(* IEC 61131-3 sources: CodesysTest/export, 96 files *)

(* ---- CheckIfHomed.st ---- *)
FUNCTION CheckIfHomed : BOOL
VAR_INPUT
	Component : IComponent;
END_VAR
VAR
	homableDevice : IHomable;
END_VAR

//	Function: CheckIfHomed()
//	Description: Helper function
//				 Pass in a component - if it has a homable motor, and is not yet homed, start homing
//	Created by: Ben Hess
//	Created Date: May 16th, 2019

IF (__QUERYINTERFACE(Component, homableDevice)) THEN
	IF homableDevice.IsHomed OR NOT Component.OptionActive THEN
		CheckIfHomed := TRUE;
		RETURN;
	ELSE
		RETURN;
	END_IF
END_IF

FUNCTION CheckIfHomed : BOOL
VAR_INPUT
	Component : IComponent;
END_VAR
VAR
	homableDevice : IHomable;
END_VAR

//	Function: CheckIfHomed()
//	Description: Helper function
//				 Pass in a component - if it has a homable motor, and is not yet homed, start homing
//	Created by: Ben Hess
//	Created Date: May 16th, 2019

IF (__QUERYINTERFACE(Component, homableDevice)) THEN
	IF homableDevice.IsHomed OR NOT Component.OptionActive THEN
		CheckIfHomed := TRUE;
		RETURN;
	ELSE
		RETURN;
	END_IF
END_IF

(* ---- EnableSimulation.st ---- *)
FUNCTION EnableSimulation : BOOL
VAR_INPUT
	device : IAllObjects;
	enableSim : BOOL;
END_VAR
VAR
	simulatable : ISimulateable;
END_VAR

//	Function: EnableSimulation()
//	Description: Helper function
//				 Pass in a device. Set simulation status if possible
//	Created by: Ben Hess
//	Created Date: June 25th, 2019

IF (__QUERYINTERFACE(device, simulatable)) THEN
	simulatable.Simulate := enableSim;
END_IF

FUNCTION EnableSimulation : BOOL
VAR_INPUT
	device : IAllObjects;
	enableSim : BOOL;
END_VAR
VAR
	simulatable : ISimulateable;
END_VAR

//	Function: EnableSimulation()
//	Description: Helper function
//				 Pass in a device. Set simulation status if possible
//	Created by: Ben Hess
//	Created Date: June 25th, 2019

IF (__QUERYINTERFACE(device, simulatable)) THEN
	simulatable.Simulate := enableSim;
END_IF

(* ---- ExhaustIfPossible.st ---- *)
FUNCTION ExhaustIfPossible : BOOL  // Attempts to exhaust SV, returns true if exhaust commanded
VAR_INPUT
	device : IAllObjects;
END_VAR
VAR
	exhaustableDevice : IExhaustable;
END_VAR

//	Function: ExhaustIfPossible()
//	Description: Helper function
//				 Pass in a device that is controlled byt a SV - exhaust if possible
//	Created by: Ben Hess
//	Created Date: June 25th, 2019

IF (__QUERYINTERFACE(device, exhaustableDevice)) THEN
	exhaustableDevice.Exhaust();
	ExhaustIfPossible := TRUE;
ELSE
	ExhaustIfPossible := FALSE;
END_IF

FUNCTION ExhaustIfPossible : BOOL  // Attempts to exhaust SV, returns true if exhaust commanded
VAR_INPUT
	device : IAllObjects;
END_VAR
VAR
	exhaustableDevice : IExhaustable;
END_VAR

//	Function: ExhaustIfPossible()
//	Description: Helper function
//				 Pass in a device that is controlled byt a SV - exhaust if possible
//	Created by: Ben Hess
//	Created Date: June 25th, 2019

IF (__QUERYINTERFACE(device, exhaustableDevice)) THEN
	exhaustableDevice.Exhaust();
	ExhaustIfPossible := TRUE;
ELSE
	ExhaustIfPossible := FALSE;
END_IF

(* ---- ExtendLPIfPossible.st ---- *)
FUNCTION ExtendLPIfPossible : BOOL
VAR_INPUT
	device : IAllObjects;
END_VAR
VAR
	extendLowPressureDevice : IExtendLowPressure;
END_VAR

//	Function: ExtendLPIfPossible()
//	Description: Helper function
//				 Pass in a device that is controlled byt a SV - extend at low pressure if possible
//	Created by: Ben Hess
//	Created Date: June 27th, 2019

IF (__QUERYINTERFACE(device, extendLowPressureDevice)) THEN
	extendLowPressureDevice.ExtendLowPressure();
	ExtendLPIfPossible := TRUE;
ELSE
	ExtendLPIfPossible := FALSE;
END_IF

FUNCTION ExtendLPIfPossible : BOOL
VAR_INPUT
	device : IAllObjects;
END_VAR
VAR
	extendLowPressureDevice : IExtendLowPressure;
END_VAR

//	Function: ExtendLPIfPossible()
//	Description: Helper function
//				 Pass in a device that is controlled byt a SV - extend at low pressure if possible
//	Created by: Ben Hess
//	Created Date: June 27th, 2019

IF (__QUERYINTERFACE(device, extendLowPressureDevice)) THEN
	extendLowPressureDevice.ExtendLowPressure();
	ExtendLPIfPossible := TRUE;
ELSE
	ExtendLPIfPossible := FALSE;
END_IF

(* ---- FirstScan.st ---- *)
FUNCTION FirstScan : DWORD
VAR_IN_OUT
	EventPrm: CmpApp.EVTPARAM_CmpApp;
END_VAR
VAR
END_VAR
// Set first scan flag from StartDone system event
Globals.firstScan := TRUE;

FUNCTION FirstScan : DWORD
VAR_IN_OUT
	EventPrm: CmpApp.EVTPARAM_CmpApp;
END_VAR
VAR
END_VAR
// Set first scan flag from StartDone system event
Globals.firstScan := TRUE;

(* ---- FN_RandomDINT.st ---- *)
FUNCTION FN_RandomDINT : DINT
VAR_INPUT
	last : DINT;
	low : DINT;
	high : DINT;
END_VAR
VAR
END_VAR

FN_RandomDINT := TO_DINT(OSCAT_BASIC.RDM(OSCAT_BASIC.FRACT(TO_REAL(last) * OSCAT_BASIC.Globale_Variablen.MATH.PI)) * (TO_REAL(high) - TO_REAL(low) + 1)) + low;

FUNCTION FN_RandomDINT : DINT
VAR_INPUT
	last : DINT;
	low : DINT;
	high : DINT;
END_VAR
VAR
END_VAR

FN_RandomDINT := TO_DINT(OSCAT_BASIC.RDM(OSCAT_BASIC.FRACT(TO_REAL(last) * OSCAT_BASIC.Globale_Variablen.MATH.PI)) * (TO_REAL(high) - TO_REAL(low) + 1)) + low;

(* ---- GetBooleanProperty.st ---- *)
// This function has been automatically generated from the project information.
{attribute 'signature_flag' := '1073741824'}
{attribute 'register_in_runtime'}
FUNCTION GetBooleanProperty : BOOL
VAR_INPUT
	stKey: WSTRING;
END_VAR
GetBooleanProperty := FALSE;

(* ---- GetCompany.st ---- *)
// This function has been automatically generated from the project information.
{attribute 'signature_flag' := '1073741824'}
{attribute 'register_in_runtime'}
FUNCTION GetCompany : WSTRING
VAR_INPUT

END_VAR
GetCompany := "Sharp Packaging";

// This function has been automatically generated from the project information.
{attribute 'signature_flag' := '1073741824'}
{attribute 'register_in_runtime'}
FUNCTION GetCompany : WSTRING
VAR_INPUT

END_VAR
GetCompany := "Sharp Packaging";

(* ---- GetLibVersion.st ---- *)
// This function has been automatically generated from the project information.
FUNCTION GetLibVersion : VERSION
VAR_INPUT

END_VAR
GetLibVersion.uiMajor := 0;
GetLibVersion.uiMinor := 2;
GetLibVersion.uiServicePack := 1;
GetLibVersion.uiPatch := 122;

// This function has been automatically generated from the project information.
FUNCTION GetLibVersion : VERSION
VAR_INPUT

END_VAR
GetLibVersion.uiMajor := 0;
GetLibVersion.uiMinor := 2;
GetLibVersion.uiServicePack := 1;
GetLibVersion.uiPatch := 122;

(* ---- GetLibVersionNumber.st ---- *)
// This function has been automatically generated from the project information.
FUNCTION GetLibVersionNumber : DWORD
VAR_INPUT

END_VAR
GetLibVersionNumber := 131450;

// This function has been automatically generated from the project information.
FUNCTION GetLibVersionNumber : DWORD
VAR_INPUT

END_VAR
GetLibVersionNumber := 131450;

(* ---- GetNumberProperty.st ---- *)
// This function has been automatically generated from the project information.
{attribute 'signature_flag' := '1073741824'}
{attribute 'register_in_runtime'}
FUNCTION GetNumberProperty : DINT
VAR_INPUT
	stKey: WSTRING;
END_VAR
GetNumberProperty := 0;

(* ---- GetTextProperty.st ---- *)
// This function has been automatically generated from the project information.
{attribute 'signature_flag' := '1073741824'}
{attribute 'register_in_runtime'}
FUNCTION GetTextProperty : WSTRING
VAR_INPUT
	stKey: WSTRING;
END_VAR
IF stKey = "Company" THEN
	GetTextProperty := "Sharp Packaging";
ELSIF stKey = "Project" THEN
	GetTextProperty := "SharpBagger";
ELSIF stKey = "Title" THEN
	GetTextProperty := "Sharp Bagger";
ELSE
	GetTextProperty := "";
END_IF

// This function has been automatically generated from the project information.
{attribute 'signature_flag' := '1073741824'}
{attribute 'register_in_runtime'}
FUNCTION GetTextProperty : WSTRING
VAR_INPUT
	stKey: WSTRING;
END_VAR
IF stKey = "Company" THEN
	GetTextProperty := "Sharp Packaging";
ELSIF stKey = "Project" THEN
	GetTextProperty := "SharpBagger";
ELSIF stKey = "Title" THEN
	GetTextProperty := "Sharp Bagger";
ELSE
	GetTextProperty := "";
END_IF

(* ---- GetTitle.st ---- *)
// This function has been automatically generated from the project information.
{attribute 'signature_flag' := '1073741824'}
{attribute 'register_in_runtime'}
FUNCTION GetTitle : WSTRING
VAR_INPUT

END_VAR
GetTitle := "Sharp Bagger";

(* ---- GetVersion.st ---- *)
// This function has been automatically generated from the project information.
{attribute 'signature_flag' := '1073741824'}
{attribute 'register_in_runtime'}
FUNCTION GetVersion : VERSION
VAR_INPUT

END_VAR
GetVersion.uiMajor := 0;
GetVersion.uiMinor := 2;
GetVersion.uiServicePack := 1;
GetVersion.uiPatch := 122;

(* ---- GetVersionProperty.st ---- *)
// This function has been automatically generated from the project information.
{attribute 'signature_flag' := '1073741824'}
{attribute 'register_in_runtime'}
FUNCTION GetVersionProperty : VERSION
VAR_INPUT
	stKey: WSTRING;
END_VAR
IF stKey = "Version" THEN
	GetVersionProperty.uiMajor := 0;
	GetVersionProperty.uiMinor := 2;
	GetVersionProperty.uiServicePack := 1;
	GetVersionProperty.uiPatch := 122;
ELSE
	GetVersionProperty.uiMajor := 0;
	GetVersionProperty.uiMinor := 0;
	GetVersionProperty.uiServicePack := 0;
	GetVersionProperty.uiPatch := 0;
END_IF

// This function has been automatically generated from the project information.
{attribute 'signature_flag' := '1073741824'}
{attribute 'register_in_runtime'}
FUNCTION GetVersionProperty : VERSION
VAR_INPUT
	stKey: WSTRING;
END_VAR
IF stKey = "Version" THEN
	GetVersionProperty.uiMajor := 0;
	GetVersionProperty.uiMinor := 2;
	GetVersionProperty.uiServicePack := 1;
	GetVersionProperty.uiPatch := 122;
ELSE
	GetVersionProperty.uiMajor := 0;
	GetVersionProperty.uiMinor := 0;
	GetVersionProperty.uiServicePack := 0;
	GetVersionProperty.uiPatch := 0;
END_IF

(* ---- HomeIfNeeded.st ---- *)
FUNCTION HomeIfNeeded : BOOL
VAR_INPUT
	Component : IComponent;
END_VAR
VAR
	homableDevice : IHomable;
END_VAR

//	Function: HomeIfNeeded()
//	Description: Helper function
//				 Pass in a component - if it has a homable motor, and is not yet homed, start homing
//	Created by: Ben Hess
//	Created Date: May 16th, 2019

IF (__QUERYINTERFACE(Component, homableDevice)) AND Component.OptionActive THEN
	IF homableDevice.IsHomed THEN
		HomeIfNeeded := TRUE;
		RETURN;
	ELSE
		homableDevice.HomeNow();
	END_IF
END_IF

(* ---- IsLibReleased.st ---- *)
// This function has been automatically generated from the project information.
FUNCTION IsLibReleased : BOOL
VAR_INPUT

END_VAR
IsLibReleased := FALSE;

(* ---- MoveRequested.st ---- *)
FUNCTION MoveRequested : BOOL
VAR_INPUT
	Component : IComponent;
END_VAR
VAR
	movableDevice : IPostHomeMove;
END_VAR

//	Function: MoveIfNeeded()
//	Description: Helper function
//				 Pass in a component - if it has a homable motor, and is not yet homed, start homing
//	Created by: Ben Hess
//	Created Date: May 16th, 2019

IF (__QUERYINTERFACE(Component, movableDevice)) AND Component.OptionActive THEN
	IF NOT movableDevice.InDesiredPosition THEN
		MoveRequested := TRUE;
		RETURN;
	ELSE
		RETURN;
	END_IF
END_IF

FUNCTION MoveRequested : BOOL
VAR_INPUT
	Component : IComponent;
END_VAR
VAR
	movableDevice : IPostHomeMove;
END_VAR

//	Function: MoveIfNeeded()
//	Description: Helper function
//				 Pass in a component - if it has a homable motor, and is not yet homed, start homing
//	Created by: Ben Hess
//	Created Date: May 16th, 2019

IF (__QUERYINTERFACE(Component, movableDevice)) AND Component.OptionActive THEN
	IF NOT movableDevice.InDesiredPosition THEN
		MoveRequested := TRUE;
		RETURN;
	ELSE
		RETURN;
	END_IF
END_IF

(* ---- MoveTimeoutCalc.st ---- *)
FUNCTION MoveTimeoutCalc : TIME
VAR_INPUT
	distance : REAL;
	velo : REAL;
	buffer : REAL;		// Buffer time to add for timeout
END_VAR
VAR
END_VAR

MoveTimeoutCalc := TO_TIME(((ABS(distance) / velo) * 1000) + buffer);

(* ---- PostHomeMoveIfNeeded.st ---- *)
FUNCTION PostHomeMoveIfNeeded : BOOL
VAR_INPUT
	Component : IComponent;
END_VAR
VAR
	movableDevice : IPostHomeMove;
END_VAR

//	Function: MoveIfNeeded()
//	Description: Helper function
//				 Pass in a component - if it has a homable motor, and is homed, and is configured for a post homing move, perform it
//	Created by: Ben Hess
//	Created Date: May 16th, 2019

IF (__QUERYINTERFACE(Component, movableDevice)) AND Component.OptionActive THEN
	IF movableDevice.InDesiredPosition THEN
		PostHomeMoveIfNeeded := TRUE;
		RETURN;
	ELSE
		movableDevice.MoveNow();
	END_IF
END_IF

(* ---- EM01_Bagger_Control_Modules.st ---- *)
FUNCTION_BLOCK EM01_Bagger_Control_Modules
VAR_INPUT
END_VAR
VAR_OUTPUT

	//simBagDelivery : FB_SimBasicBagDelivery(name := 'Sim Bag Delivery'):= (enable := TRUE, installed := TRUE);
	//simPrinter : FB_SimBasicPrinter(name := 'Sim Printer'):= (enable := TRUE, installed := TRUE);
	//simVacuumCups : FB_SimBasicVacuum(name := 'Sim Vac Cups') := (_optionEnabled := TRUE, _optionInstalled := TRUE);
	vacuumCups : FB_PneumaticVacuumCups(name := 'Pneumatic Vacuum Cups') := (_optionEnabled := TRUE, _optionInstalled := TRUE);
	simLoadPlate : FB_SimBasicLoadPlate(name := 'Sim Load Plate') := (_optionEnabled := TRUE, _optionInstalled := TRUE);
	simExitConveyor : FB_SimBasicExitConveyor(name := 'Sim Exit Conveyor') := (_optionEnabled := TRUE, _optionInstalled := TRUE);

	standardSealBar : FB_PneumaticSealer(name := 'Pneumatic Seal Bar') := (_optionEnabled := TRUE, _optionInstalled := TRUE);
	standardBagOpenFingersWithSensors : FB_PneuBagOpenFingersWithSensorsOLD(name := 'Standard Bag Open Fingers') := (_optionEnabled := TRUE, _optionInstalled := TRUE);
	pneumaticPressureBar : FB_PneuPBarWithAdjPass(name := 'Pneumatic Pressure Bar') := (_optionEnabled := TRUE, _optionInstalled := TRUE);
	motorizedSealFlatteners : FB_MotorizedSealFlatteners(name := 'Motorized Seal Flatteners') := (_optionEnabled := TRUE, _optionInstalled := TRUE);

	passthroughMotor : FB_SimMotor;
	msfHorizontalMotor : FB_SimMotor;
	bagOpenFingersActuator : FB_PneumaticVerticalActuator(name := 'Bag Open Fingers Actuator');
	sealFlattenerVertAxisActuator : FB_PneumaticVerticalActuator(name := 'Seal Flat Pneu Vert Axis Actuator');

	bagDelivery : FB_Pro18BagDelivery(name := 'Bag Delivery') := (_optionEnabled := TRUE, _optionInstalled := TRUE);
	bagDeliveryFrontMotor : FB_SimMotor;

	labelPrinter : FB_Pro18ZebraPrinter(name := 'Zebra Label Printer') := (_optionEnabled := TRUE, _optionInstalled := TRUE);
	printHeadActuator : FB_PneumaticVerticalActuator(name := 'Print Head Actuator');
END_VAR

VAR
END_VAR

// simBagDelivery(
// 	enable:= ,
// 	installed:= ,
// 	active=> ,
// 	feedSpeed:= HMI.data.bagForwardSpeed,
// 	reverseSpeed:= HMI.data.bagReverseSpeed,
// 	printSpeed:= HMI.data.printSpeed,
// 	printLength:= HMI.data.printLength,
// 	bagLength:= HMI.data.bagLength,
// 	reverseLength:= 2.0,
// 	printOffset:= HMI.data.printOffset);

//sealFlattenerPneuVerticalAxis(cylinder := sealFlattenerVertAxisActuator);

simExitConveyor(_optionActive=> );

simLoadPlate(_optionActive=> , loadPlateDwell:= HMI.data.loadPlateDwell);

passthroughMotor(simFault := UN00_Globals.simFaults.passthroughMotorFault);

pneumaticPressureBar(
	_optionActive=> ,
	simulateIO:= HMI.data.simulateAllIO,
	passthroughMotor:= passthroughMotor,
	cylinder := Devices.pressureBarSolenoidValve,
	ptVelo:= ,
	ptAccel:= ,
	ptDecel:= ,
	homeTimeoutSetting:= ,
	passthroughSetting := HMI.data.passthroughSetting,
	failedToClose=> ,
	failedToOpen=> ,
	failedToHome=> ,
	pressureBarObstructed=> ,
	motorFault=> ,
	failedToMovePassthrough=> ,
	actualPassthrough=> HMI.data.passthroughActual,
	PressureBarClosedSensor:= IO.iPressureBarRetracted,
	PressureBarOpenSensor:= IO.iPressureBarExtended,
	ObstructionSensor := IO.iPressureBarNotObstructed);

printHeadActuator(cylinder := Devices.printHeadSolenoidValve);
labelPrinter(
	_optionActive=> ,
	simulateIO:= HMI.data.simulateAllIO,
	printSpeed:= HMI.data.printSpeed,
	printLength:= HMI.data.printLength,
	printHead:= printHeadActuator,
	dataReadyInput:= IO.iPrinterDataReady,
	serviceRequiredInput:= IO.iPrinterServiceRequired,
	ribbonLowInput:= IO.iPrinterRibbonOut,
	endOfPrintInput:= IO.iPrinterEndOfPrint,
	printHeadDebounceSetpoint:= ,
	serviceRequired=> ,
	ribbonLow=> ,
	startPrintOutput:= IO.oPrinterStartPrint,
	ribbonUnwindRunOutput:= IO.oRunRibbonUnwindMotor);

standardSealBar(
	_optionActive=> ,
	simulateIO:= HMI.data.simulateAllIO,
	sealDwell:= HMI.data.sealBarDwell,
	cylinder:= Devices.sealBarSolenoidValve);

vacuumCups(_optionActive=>, vacGenerator := Devices.vacuumSolenoidValve);
bagOpenFingersActuator(cylinder:= Devices.bagOpenFingersSolenoidValve);
standardBagOpenFingersWithSensors(
	simulateIO:= HMI.data.simulateAllIO,
	simMissedBag:= UN00_Globals.simFaults.failedToGrabBagLeftFinger,
	_optionActive=> ,
	delayToGrabSetting:= HMI.data.grabBagDelay,
	delayToCheckBagPresentSetting:= HMI.data.checkForBagOpenDelay,
	delayToClearSetting:= HMI.data.bagClearedFromFingersDelay,
	fingerActuators := bagOpenFingersActuator,
	BagPresentSensorLeft:= IO.iBagOpenFingersLeftBagPresent,
	BagPresentSensorRight:= IO.iBagOpenFingersRightBagPresent);

sealFlattenerVertAxisActuator(solenoid0=> , solenoid1=> , cylinder:= Devices.sealFlattenersVertAxisSolenoidValve);
msfHorizontalMotor();
motorizedSealFlatteners(
	_optionActive=> ,
	clearanceDwellSetting:= HMI.data.bagDropClearanceDwell,
	bagWidth:= HMI.data.bagWidth,
	horizVelo:= ,
	horizAccel:= ,
	horizDecel:= ,
	bagHoldingCurrent:= ,
	sealCurrentAddition:= ,
	homeTimeoutSetting:= ,
	maximumPosition:= ,
	miniumumPosition:= ,
	clearanceOffset:= ,
	msfHorizActualPosition=> ,
	horizontalFailedToMove=> ,
	horizontalFailedToHome=> ,
	motorFault=> ,
	verticalAxis:= sealFlattenerVertAxisActuator,
	horizontalAxis:= msfHorizontalMotor);

	bagDeliveryFrontMotor();
	bagDelivery(
	simulateIO := HMI.data.simulateAllIO,
	_optionActive=> ,
	printer:= labelPrinter,
	bagLength:= HMI.data.bagLength,
	feedSpeed:= TO_REAL(HMI.data.bagForwardSpeed),
	reverseSpeed:= TO_REAL(HMI.data.bagReverseSpeed),
	printSpeed:= ,
	printOffset:= ,
	printLength:= ,
	maxReverseSetpoint:= ,
	sealOffset:= ,
	distanceFromSealBarToBagEdge:= ,
	distanceFromNipToBagEdge:= ,
	bagPhotoeyeInput:= IO.iBagPhotoeyeClear,
	trapezoidalPercent:= ,
	bagDeliveryFailedToMove=> ,
	bagFailedToSeparate=> ,
	bagDeliveryMotor:= bagDeliveryFrontMotor);

FUNCTION_BLOCK EM01_Bagger_Control_Modules
VAR_INPUT
END_VAR
VAR_OUTPUT

	//simBagDelivery : FB_SimBasicBagDelivery(name := 'Sim Bag Delivery'):= (enable := TRUE, installed := TRUE);
	//simPrinter : FB_SimBasicPrinter(name := 'Sim Printer'):= (enable := TRUE, installed := TRUE);
	//simVacuumCups : FB_SimBasicVacuum(name := 'Sim Vac Cups') := (_optionEnabled := TRUE, _optionInstalled := TRUE);
	vacuumCups : FB_PneumaticVacuumCups(name := 'Pneumatic Vacuum Cups') := (_optionEnabled := TRUE, _optionInstalled := TRUE);
	simLoadPlate : FB_SimBasicLoadPlate(name := 'Sim Load Plate') := (_optionEnabled := TRUE, _optionInstalled := TRUE);
	simExitConveyor : FB_SimBasicExitConveyor(name := 'Sim Exit Conveyor') := (_optionEnabled := TRUE, _optionInstalled := TRUE);

	standardSealBar : FB_PneumaticSealer(name := 'Pneumatic Seal Bar') := (_optionEnabled := TRUE, _optionInstalled := TRUE);
	standardBagOpenFingersWithSensors : FB_PneuBagOpenFingersWithSensorsOLD(name := 'Standard Bag Open Fingers') := (_optionEnabled := TRUE, _optionInstalled := TRUE);
	pneumaticPressureBar : FB_PneuPBarWithAdjPass(name := 'Pneumatic Pressure Bar') := (_optionEnabled := TRUE, _optionInstalled := TRUE);
	motorizedSealFlatteners : FB_MotorizedSealFlatteners(name := 'Motorized Seal Flatteners') := (_optionEnabled := TRUE, _optionInstalled := TRUE);

	passthroughMotor : FB_SimMotor;
	msfHorizontalMotor : FB_SimMotor;
	bagOpenFingersActuator : FB_PneumaticVerticalActuator(name := 'Bag Open Fingers Actuator');
	sealFlattenerVertAxisActuator : FB_PneumaticVerticalActuator(name := 'Seal Flat Pneu Vert Axis Actuator');

	bagDelivery : FB_Pro18BagDelivery(name := 'Bag Delivery') := (_optionEnabled := TRUE, _optionInstalled := TRUE);
	bagDeliveryFrontMotor : FB_SimMotor;

	labelPrinter : FB_Pro18ZebraPrinter(name := 'Zebra Label Printer') := (_optionEnabled := TRUE, _optionInstalled := TRUE);
	printHeadActuator : FB_PneumaticVerticalActuator(name := 'Print Head Actuator');
END_VAR

VAR
END_VAR

// simBagDelivery(
// 	enable:= ,
// 	installed:= ,
// 	active=> ,
// 	feedSpeed:= HMI.data.bagForwardSpeed,
// 	reverseSpeed:= HMI.data.bagReverseSpeed,
// 	printSpeed:= HMI.data.printSpeed,
// 	printLength:= HMI.data.printLength,
// 	bagLength:= HMI.data.bagLength,
// 	reverseLength:= 2.0,
// 	printOffset:= HMI.data.printOffset);

//sealFlattenerPneuVerticalAxis(cylinder := sealFlattenerVertAxisActuator);

simExitConveyor(_optionActive=> );

simLoadPlate(_optionActive=> , loadPlateDwell:= HMI.data.loadPlateDwell);

passthroughMotor(simFault := UN00_Globals.simFaults.passthroughMotorFault);

pneumaticPressureBar(
	_optionActive=> ,
	simulateIO:= HMI.data.simulateAllIO,
	passthroughMotor:= passthroughMotor,
	cylinder := Devices.pressureBarSolenoidValve,
	ptVelo:= ,
	ptAccel:= ,
	ptDecel:= ,
	homeTimeoutSetting:= ,
	passthroughSetting := HMI.data.passthroughSetting,
	failedToClose=> ,
	failedToOpen=> ,
	failedToHome=> ,
	pressureBarObstructed=> ,
	motorFault=> ,
	failedToMovePassthrough=> ,
	actualPassthrough=> HMI.data.passthroughActual,
	PressureBarClosedSensor:= IO.iPressureBarRetracted,
	PressureBarOpenSensor:= IO.iPressureBarExtended,
	ObstructionSensor := IO.iPressureBarNotObstructed);

printHeadActuator(cylinder := Devices.printHeadSolenoidValve);
labelPrinter(
	_optionActive=> ,
	simulateIO:= HMI.data.simulateAllIO,
	printSpeed:= HMI.data.printSpeed,
	printLength:= HMI.data.printLength,
	printHead:= printHeadActuator,
	dataReadyInput:= IO.iPrinterDataReady,
	serviceRequiredInput:= IO.iPrinterServiceRequired,
	ribbonLowInput:= IO.iPrinterRibbonOut,
	endOfPrintInput:= IO.iPrinterEndOfPrint,
	printHeadDebounceSetpoint:= ,
	serviceRequired=> ,
	ribbonLow=> ,
	startPrintOutput:= IO.oPrinterStartPrint,
	ribbonUnwindRunOutput:= IO.oRunRibbonUnwindMotor);

standardSealBar(
	_optionActive=> ,
	simulateIO:= HMI.data.simulateAllIO,
	sealDwell:= HMI.data.sealBarDwell,
	cylinder:= Devices.sealBarSolenoidValve);

vacuumCups(_optionActive=>, vacGenerator := Devices.vacuumSolenoidValve);
bagOpenFingersActuator(cylinder:= Devices.bagOpenFingersSolenoidValve);
standardBagOpenFingersWithSensors(
	simulateIO:= HMI.data.simulateAllIO,
	simMissedBag:= UN00_Globals.simFaults.failedToGrabBagLeftFinger,
	_optionActive=> ,
	delayToGrabSetting:= HMI.data.grabBagDelay,
	delayToCheckBagPresentSetting:= HMI.data.checkForBagOpenDelay,
	delayToClearSetting:= HMI.data.bagClearedFromFingersDelay,
	fingerActuators := bagOpenFingersActuator,
	BagPresentSensorLeft:= IO.iBagOpenFingersLeftBagPresent,
	BagPresentSensorRight:= IO.iBagOpenFingersRightBagPresent);

sealFlattenerVertAxisActuator(solenoid0=> , solenoid1=> , cylinder:= Devices.sealFlattenersVertAxisSolenoidValve);
msfHorizontalMotor();
motorizedSealFlatteners(
	_optionActive=> ,
	clearanceDwellSetting:= HMI.data.bagDropClearanceDwell,
	bagWidth:= HMI.data.bagWidth,
	horizVelo:= ,
	horizAccel:= ,
	horizDecel:= ,
	bagHoldingCurrent:= ,
	sealCurrentAddition:= ,
	homeTimeoutSetting:= ,
	maximumPosition:= ,
	miniumumPosition:= ,
	clearanceOffset:= ,
	msfHorizActualPosition=> ,
	horizontalFailedToMove=> ,
	horizontalFailedToHome=> ,
	motorFault=> ,
	verticalAxis:= sealFlattenerVertAxisActuator,
	horizontalAxis:= msfHorizontalMotor);

	bagDeliveryFrontMotor();
	bagDelivery(
	simulateIO := HMI.data.simulateAllIO,
	_optionActive=> ,
	printer:= labelPrinter,
	bagLength:= HMI.data.bagLength,
	feedSpeed:= TO_REAL(HMI.data.bagForwardSpeed),
	reverseSpeed:= TO_REAL(HMI.data.bagReverseSpeed),
	printSpeed:= ,
	printOffset:= ,
	printLength:= ,
	maxReverseSetpoint:= ,
	sealOffset:= ,
	distanceFromSealBarToBagEdge:= ,
	distanceFromNipToBagEdge:= ,
	bagPhotoeyeInput:= IO.iBagPhotoeyeClear,
	trapezoidalPercent:= ,
	bagDeliveryFailedToMove=> ,
	bagFailedToSeparate=> ,
	bagDeliveryMotor:= bagDeliveryFrontMotor);

(* ---- EM01_BaggerHead.st ---- *)
FUNCTION_BLOCK EM01_BaggerHead EXTENDS FB_PackMLStates IMPLEMENTS IEM01_BaggerHead
VAR_INPUT
	(*Comnponents*)
	bagOpenFingers : IBagOpenFingers;
	sealFlatteners : ISealFlatteners;
	sealer : ISealer;
	pressureBar : IPressureBar;
	printer : IPrinter;
	bagDelivery : IBagDelivery;
	vacuumBagOpen : IVacuumBagOpen;

	(*Options and settings*)
	bagOpenAssistEnabled : BOOL;		// Bag Open Assist Option Enabled from HMI
	bagOpenSensorEnabled : BOOL;		// Bag Open Sensors Enabled from HMI
	separateBeforeSealEnabled : BOOL;	// Separate before Seal Option Enabled from HMI
	bagOpenRetrySetting : UINT;
	newJobLoaded : BOOL;
	vacuumDwell : TIME;
END_VAR
VAR_OUTPUT
	baggerCycleActive : BOOL;
	bagOpenRetryCount : UINT;
	failedToOpenBag : FB_Fault(name := CONCAT(_prefix,'Failed to Open Bag'));
END_VAR
VAR
	_startCycle : BOOL;
	_readyToAcceptProduct : BOOL;
END_VAR

PROPERTY ReadyForProduct : BOOL

METHOD StartCycle

_startCycle := TRUE;

PROPERTY StartCycleRequest : BOOL

PROPERTY CurrentBagOpenRetryCount : UINT

FUNCTION_BLOCK EM01_BaggerHead EXTENDS FB_PackMLStates IMPLEMENTS IEM01_BaggerHead
VAR_INPUT
	(*Comnponents*)
	bagOpenFingers : IBagOpenFingers;
	sealFlatteners : ISealFlatteners;
	sealer : ISealer;
	pressureBar : IPressureBar;
	printer : IPrinter;
	bagDelivery : IBagDelivery;
	vacuumBagOpen : IVacuumBagOpen;

	(*Options and settings*)
	bagOpenAssistEnabled : BOOL;		// Bag Open Assist Option Enabled from HMI
	bagOpenSensorEnabled : BOOL;		// Bag Open Sensors Enabled from HMI
	separateBeforeSealEnabled : BOOL;	// Separate before Seal Option Enabled from HMI
	bagOpenRetrySetting : UINT;
	newJobLoaded : BOOL;
	vacuumDwell : TIME;
END_VAR
VAR_OUTPUT
	baggerCycleActive : BOOL;
	bagOpenRetryCount : UINT;
	failedToOpenBag : FB_Fault(name := CONCAT(_prefix,'Failed to Open Bag'));
END_VAR
VAR
	_startCycle : BOOL;
	_readyToAcceptProduct : BOOL;
END_VAR

PROPERTY ReadyForProduct : BOOL

METHOD StartCycle

_startCycle := TRUE;

PROPERTY StartCycleRequest : BOOL

PROPERTY CurrentBagOpenRetryCount : UINT

(* ---- EM01_BaggerHead_Automode.st ---- *)
FUNCTION_BLOCK EM01_BaggerHead_Automode EXTENDS FB_PackMLStates
VAR_INPUT
	infeed : IEM00_Product_Infeed;
	discharge : IEM02_Discharge;
END_VAR
VAR_OUTPUT
	state : HEAD_STATES;
    sealAndSeparateSubState : SEAL_SEPARATE_STATES;
    releaseAndFeedSubState : RELEASE_FEED_STATES;
    bagOpenSubState : BAG_OPEN_ASSIST_STATES;
	currentBaggerState : STRING;
END_VAR
VAR
	cycleTimer : TON() := (PT := T#1000S);
	cycleTime : REAL;
	resetTriggered : BOOL;
	resettingState : INT;
	vacuumDwellTimer : TON;
END_VAR
VAR_IN_OUT
	bagger : EM01_BaggerHead;
END_VAR

//	Function Block: EM01_Bagger_Automode
//	Description: This is an implementation of a bagger in Auto Mode (normal operation) using the PackML standard.
//				 Each method is a PackML state.
//	Created by: Ben Hess
//	Created Date: Tuesday, March 26, 2019

METHOD Stopping

_stoppingDone := TRUE;

METHOD Stopped

_clearingDone := FALSE;
_stoppingDone := FALSE;
resetTriggered := FALSE;

METHOD Resetting

state := HEAD_STATES.Idle;
sealAndSeparateSubState := SEAL_SEPARATE_STATES.Idle;
releaseAndFeedSubState := RELEASE_FEED_STATES.Idle;
bagOpenSubState := BAG_OPEN_ASSIST_STATES.Idle;

CASE resettingState OF
	0:	// Clear PackML state bits and Home everything that needs homing
		_clearingDone := FALSE;
		_completingDone := FALSE;
		_holdingDone := FALSE;
		_resettingDone := FALSE;
		_startingDone := FALSE;
		_unholdingDone := FALSE;
		_stoppingDone := FALSE;

		vacuumDwellTimer.IN := FALSE;

		bagger.bagDelivery.Reset();
		HomeIfNeeded(bagger.pressureBar);
		HomeIfNeeded(bagger.sealFlatteners);
		resettingState := 1;

	1:	// Move everything into place to start machine
		IF CheckIfHomed(bagger.pressureBar) THEN
			PostHomeMoveIfNeeded(bagger.pressureBar);
			resettingState := 2;
		END_IF

	2:	// Once everything is moved into position and ready move on
		IF bagger.pressureBar.Ready OR NOT bagger.pressureBar.OptionActive THEN
			_resettingDone := TRUE;
		END_IF

END_CASE

METHOD Idle

_resettingDone := FALSE;
resettingState := 0;
resetTriggered := FALSE;

METHOD Starting

IF NOT _startingDone THEN
	bagger.pressureBar.Open();
	bagger.bagOpenFingers.ReleaseBag();
	bagger.sealFlatteners.ToBagFeed();
	_startingDone := TRUE;
END_IF

METHOD Executing

//	Method: EM01_Bagger_Automode.Executing()
//	Description: Executing is the state in which the machine is producing bags.  In this state, the bagger is homed and ready to initiate a cycle any time.
//				 In normal operation, the machine should be in this state most of the time
//				 The logic below is generic and coded to interfaces for each component
//	Created by: Ben Hess
//	Created Date: Tuesday, March 26, 2019

IF NOT __ISVALIDREF(bagger) THEN
	RETURN;
END_IF

// Clear starting done status because if we're here starting state is complete.
_startingDone := FALSE;

// Run Cycle timer for machine cycle
cycleTimer();
vacuumDwellTimer(PT := bagger.vacuumDwell);
// State machine for overall head states
CASE state OF
    HEAD_STATES.Idle :                              // Start cycle
                                                    IF bagger.StartCycleRequest THEN
														bagger.StartCycleRequest := FALSE;
														cycleTimer.IN := TRUE;
														_logger.AddLogItem('Cycle Started');
														SetHeadState(HEAD_STATES.SealAndSeparateBag);
													END_IF

													IF MoveRequested (bagger.pressureBar) THEN
														SetHeadState(HEAD_STATES.MovePassthrough);
													END_IF

	HEAD_STATES.MovePassthrough : 					//
													PostHomeMoveIfNeeded(bagger.pressureBar);
													SetHeadState(HEAD_STATES.MovingPassthrough);

    HEAD_STATES.MovingPassthrough :                 //
													IF NOT MoveRequested (bagger.pressureBar) THEN
														SetHeadState(HEAD_STATES.MovedPassthrough);
													END_IF

	HEAD_STATES.MovedPassthrough : 					//
													SetHeadState(HEAD_STATES.Idle);

    HEAD_STATES.SealAndSeparateBag :                // Begin Seal and Separate State machine
                                                    SetSealSeparateState(SEAL_SEPARATE_STATES.MoveJawIn);
													SetHeadState(HEAD_STATES.SealingAndSeparatingBag);

    HEAD_STATES.SealingAndSeparatingBag :          //
													IF sealAndSeparateSubState = SEAL_SEPARATE_STATES.Done THEN
														SetHeadState(HEAD_STATES.SealedAndSeparatedBag);
														SetSealSeparateState(SEAL_SEPARATE_STATES.Idle);
                                                    END_IF

    HEAD_STATES.SealedAndSeparatedBag :             //
													SetHeadState(HEAD_STATES.ReleaseAndFeedBag);

    HEAD_STATES.ReleaseAndFeedBag :                 // Open the jaw and release the bag
													SetReleaseFeedState(RELEASE_FEED_STATES.MoveJawOutAndFeedBag);
                                                    SetHeadState(HEAD_STATES.ReleasingAndFeedingBag);

    HEAD_STATES.ReleasingAndFeedingBag :            //
                                                    IF releaseAndFeedSubState = RELEASE_FEED_STATES.Done THEN
                                                        SetHeadState(HEAD_STATES.ReleasedAndFedBag);
                                                        SetReleaseFeedState(RELEASE_FEED_STATES.Idle);
                                                    END_IF

    HEAD_STATES.ReleasedAndFedBag :                 // Start opening bag if bag open assist is enabled, otherwise end cycle now
													IF bagger.bagOpenAssistEnabled THEN
														SetHeadState(HEAD_STATES.OpenBag);
													ELSE
														SetHeadState(HEAD_STATES.OpenedBag);
													END_IF

    HEAD_STATES.OpenBag :                            // Close jaw to grab the bag
                                                    SetBagOpenState(BAG_OPEN_ASSIST_STATES.MoveJawIn);
                                                    SetHeadState(HEAD_STATES.OpeningBag);

    HEAD_STATES.OpeningBag :                        // Open jaw and grab onto the bag.  Feed a new bag out if missed
                                                    IF bagOpenSubState = BAG_OPEN_ASSIST_STATES.Done THEN
                                                        SetHeadState(HEAD_STATES.OpenedBag);
                                                        SetBagOpenState(BAG_OPEN_ASSIST_STATES.Idle);
													ELSIF bagOpenSubState = BAG_OPEN_ASSIST_STATES.FeedNewBag THEN
														SetHeadState(HEAD_STATES.SealAndSeparateBag);
														SetBagOpenState(BAG_OPEN_ASSIST_STATES.Idle);
                                                    END_IF

    HEAD_STATES.OpenedBag :                         // End cycle
                                                    SetHeadState(HEAD_STATES.Idle);
													cycleTime := (TIME_TO_REAL(cycleTimer.ET) / 1000);
													cycleTimer.IN := FALSE;
													_logger.AddLogItem(CONCAT('Cycle Complete in ',TO_STRING(cycleTime)));

    //HEAD_STATES.Fault :

END_CASE

CASE sealAndSeparateSubState OF
    //SEAL_SEPARATE_STATES.Idle :

    SEAL_SEPARATE_STATES.MoveJawIn :                // Perform actions as enabled - close jaw and move flatteners out. If jaw is disabled then go right to reverse bag
                                                    IF bagger.sealFlatteners.OptionActive THEN
														bagger.sealFlatteners.ToSeal();
													END_IF
                                                    bagger.pressureBar.Close();
													SetSealSeparateState(SEAL_SEPARATE_STATES.MovingJawIn);

    SEAL_SEPARATE_STATES.MovingJawIn :              // If Jaw is in and flatteners out then move on
                                                   	IF (NOT bagger.sealFlatteners.OptionActive OR bagger.sealFlatteners.InPosition)
														AND bagger.pressureBar.IsFullyClosed THEN
															SetSealSeparateState(SEAL_SEPARATE_STATES.MovedJawIn);
                                                    END_IF

    SEAL_SEPARATE_STATES.MovedJawIn :               // Seal bag now if separate before seal option selected
													IF NOT bagger.separateBeforeSealEnabled THEN
														bagger.sealer.BeginSealing();
													END_IF
													SetSealSeparateState(SEAL_SEPARATE_STATES.ReverseBag);

    SEAL_SEPARATE_STATES.ReverseBag :               // Start reversing bag to seal
													bagger.bagDelivery.ReverseToSeparate();
													SetSealSeparateState(SEAL_SEPARATE_STATES.ReversingBag);

    SEAL_SEPARATE_STATES.ReversingBag :             //
                                                    IF bagger.bagDelivery.BagSeparated
														AND (bagger.sealer.SealComplete OR bagger.separateBeforeSealEnabled)
                                                        THEN
															SetSealSeparateState(SEAL_SEPARATE_STATES.Reversedbag);
                                                    END_IF

    SEAL_SEPARATE_STATES.Reversedbag :              //
                                                    IF bagger.separateBeforeSealEnabled THEN
														SetSealSeparateState(SEAL_SEPARATE_STATES.SealBag);
													ELSE
														SetSealSeparateState(SEAL_SEPARATE_STATES.Done);
													END_IF

	SEAL_SEPARATE_STATES.SealBag:
													bagger.sealer.BeginSealing();
													SetSealSeparateState(SEAL_SEPARATE_STATES.SealingBag);

	SEAL_SEPARATE_STATES.SealingBag:				//
													IF bagger.sealer.SealComplete THEN
														SetSealSeparateState(SEAL_SEPARATE_STATES.Done);
													END_IF

    //SEAL_SEPARATE_STATES.Done :                   //

    //SEAL_SEPARATE_STATES.Fault :					//
END_CASE

CASE releaseAndFeedSubState OF
    //RELEASE_FEED_STATES.Idle :                    //

    RELEASE_FEED_STATES.MoveJawOutAndFeedBag :
													bagger.bagOpenFingers.ReleaseBag();
													bagger.sealFlatteners.ToBagFeed();
													bagger.pressureBar.Open();

													discharge.TakeAwayBag(THIS^);
													releaseAndFeedSubState := RELEASE_FEED_STATES.WaitForOKFromDischarge;
													// If printer is enabled then perform printer operation of bag delivery, otherwise just feed new bag out.
													IF NOT bagger.printer.OptionActive THEN
														bagger.bagDelivery.FeedBagOut();
														SetReleaseFeedState(RELEASE_FEED_STATES.MovingJawOutAndFeedingBag);
													ELSE
														SetReleaseFeedState(RELEASE_FEED_STATES.WaitForPrinter);
													END_IF

    RELEASE_FEED_STATES.WaitForOKFromDischarge :   	// Wait for EM02 - Discharge to give OK to feed bag signal
													IF discharge.OKToFeedBag THEN
														IF NOT bagger.printer.OptionActive THEN
															bagger.bagDelivery.FeedBagOut();
															SetReleaseFeedState(RELEASE_FEED_STATES.MovingJawOutAndFeedingBag);
														ELSE
															SetReleaseFeedState(RELEASE_FEED_STATES.WaitForPrinter);
														END_IF
													END_IF

    RELEASE_FEED_STATES.WaitForPrinter :            // Data Ready means the printer has a label and we're all set to print
                                                    IF bagger.printer.HasLabel THEN
														SetReleaseFeedState(RELEASE_FEED_STATES.FeedToOffset);
                                                    END_IF

    RELEASE_FEED_STATES.FeedToOffset :              // Start feeding to the print offset
                                                    bagger.bagDelivery.FeedToPrintOffset();
													SetReleaseFeedState(RELEASE_FEED_STATES.FeedingToOffset);

    RELEASE_FEED_STATES.FeedingToOffset :            // Once offset done start printing
                                                    IF bagger.bagDelivery.ReadyForPrint THEN
														SetReleaseFeedState(RELEASE_FEED_STATES.StartPrinting);
                                                    END_IF

    RELEASE_FEED_STATES.StartPrinting :             // Printer starts print cycle and bag delivery starts moving at print speed
													bagger.printer.BeginPrinting();
													bagger.bagDelivery.FeedAtPrintSpeed();
													SetReleaseFeedState(RELEASE_FEED_STATES.Printing);

    //RELEASE_FEED_STATES.SendPrintSignal:            //

    RELEASE_FEED_STATES.Printing :                  // Wait for print to finish
                                                    IF bagger.printer.PrintDone THEN
														SetReleaseFeedState(RELEASE_FEED_STATES.StopPrinting);
                                                    END_IF

    RELEASE_FEED_STATES.StopPrinting :              // Tell bag delivery it's okay to feed out the rest of the bag and the printer that it can prep itself for the next print
                                                    bagger.bagDelivery.FeedBagOut();
													SetReleaseFeedState(RELEASE_FEED_STATES.MovingJawOutAndFeedingBag);

    RELEASE_FEED_STATES.MovingJawOutAndFeedingBag : //
													IF (bagger.sealFlatteners.InPosition OR NOT bagger.sealFlatteners.OptionActive)
                                                        AND bagger.pressureBar.IsFullyOpen
														AND bagger.bagDelivery.BagFeedDone
                                                        THEN
															SetReleaseFeedState(RELEASE_FEED_STATES.MovedJawOutAndFedBag);
                                                    END_IF

    RELEASE_FEED_STATES.MovedJawOutAndFedBag :
													SetReleaseFeedState(RELEASE_FEED_STATES.Done);
    //RELEASE_FEED_STATES.Done :
    //RELEASE_FEED_STATES.Fault :
END_CASE

CASE bagOpenSubState OF
    BAG_OPEN_ASSIST_STATES.Idle :                    //

    BAG_OPEN_ASSIST_STATES.MoveJawIn :                // Close jaw against bag. In the future we may also start vacuum here
                                                    bagger.pressureBar.Close();
													SetBagOpenState(BAG_OPEN_ASSIST_STATES.MovingJawIn);

    BAG_OPEN_ASSIST_STATES.MovingJawIn :            // Move on once jaw is closed
                                                    IF bagger.pressureBar.IsFullyClosed THEN
														IF bagger.vacuumBagOpen.OptionActive THEN
															bagger.vacuumBagOpen.StartVacuum();
														END_IF
														SetBagOpenState(BAG_OPEN_ASSIST_STATES.MovedJawIn);
                                                    END_IF

    BAG_OPEN_ASSIST_STATES.MovedJawIn :             // Hold onto the bag with vacuum to build suction
													vacuumDwellTimer.IN := TRUE;
													IF (vacuumDwellTimer.Q OR NOT bagger.vacuumBagOpen.OptionActive) THEN
														vacuumDwellTimer.IN := FALSE;
														SetBagOpenState(BAG_OPEN_ASSIST_STATES.MoveJawOut);
													END_IF

    BAG_OPEN_ASSIST_STATES.MoveJawOut :             // Open the jaw and move seal flatteners in and to bag holding
                                                    bagger.pressureBar.Open();
													SetBagOpenState(BAG_OPEN_ASSIST_STATES.MovingJawOutAndGrab);

    BAG_OPEN_ASSIST_STATES.MovingJawOutAndGrab :    	//
														IF bagger.bagOpenFingers.OptionActive THEN
															bagger.bagOpenFingers.GrabBag();
															IF bagger.bagOpenSensorEnabled THEN
																SetBagOpenState(BAG_OPEN_ASSIST_STATES.CheckForSuccessfulBagGrab);
															ELSE
																SetBagOpenState(BAG_OPEN_ASSIST_STATES.BagOpened);
															END_IF
														ELSE
															SetBagOpenState(BAG_OPEN_ASSIST_STATES.BagOpened);
														END_IF

	BAG_OPEN_ASSIST_STATES.CheckForSuccessfulBagGrab : 	//
														IF bagger.CurrentBagOpenRetryCount < bagger.bagOpenRetrySetting THEN
															IF bagger.bagOpenFingers.BagGrabbed THEN
																SetBagOpenState(BAG_OPEN_ASSIST_STATES.BagOpened);
															ELSIF bagger.bagOpenFingers.BagMissed THEN
																SetBagOpenState(BAG_OPEN_ASSIST_STATES.BagFailedToOpen);
															END_IF
														ELSE
															SetBagOpenState(BAG_OPEN_ASSIST_STATES.MovingJawOutAfterGrab);
														END_IF

	BAG_OPEN_ASSIST_STATES.BagFailedToOpen :			//
														bagger.bagOpenFingers.ReleaseBag();
														bagger.CurrentBagOpenRetryCount := bagger.CurrentBagOpenRetryCount + 1;
														IF bagger.CurrentBagOpenRetryCount < bagger.bagOpenRetrySetting THEN
															SetBagOpenState(BAG_OPEN_ASSIST_STATES.MoveJawIn);
														ELSE
															SetBagOpenState(BAG_OPEN_ASSIST_STATES.MovingJawOutAfterGrab);
															bagger.CurrentBagOpenRetryCount := 0;
															bagger.failedToOpenBag.Trigger();
														END_IF

	BAG_OPEN_ASSIST_STATES.BagOpened :					//
														bagger.vacuumBagOpen.StopVacuum();
                                                    	bagger.sealFlatteners.BagIsOpen();
														bagger.CurrentBagOpenRetryCount := 0;
// 														HMIData.bagsMade.Increment();
// 														HMIData.airFilterClean.Increment();
// 														HMIData.baggerCycles.Increment();
														SetBagOpenState(BAG_OPEN_ASSIST_STATES.MovingJawOutAfterGrab);

    BAG_OPEN_ASSIST_STATES.MovingJawOutAfterGrab :		//
														IF bagger.pressureBar.IsFullyOpen
															AND (bagger.sealFlatteners.InPosition OR NOT bagger.sealFlatteners.OptionActive)
															THEN
																SetBagOpenState(BAG_OPEN_ASSIST_STATES.MovedJawOut);
														END_IF

	BAG_OPEN_ASSIST_STATES.MovedJawOut :            	//

														SetBagOpenState(BAG_OPEN_ASSIST_STATES.Done);

	//BAG_OPEN_ASSIST_STATES.FeedNewBag :   				//

    //BAG_OPEN_ASSIST_STATES.Done :                    	//

    //BAG_OPEN_ASSIST_STATES.Fault :                    //

END_CASE

METHOD Aborting

IF NOT _abortingDone THEN
	_clearingDone := FALSE;
	_completingDone := FALSE;
	_holdingDone := FALSE;
	_resettingDone := FALSE;
	_startingDone := FALSE;
	_unholdingDone := FALSE;
	_stoppingDone := FALSE;
	resetTriggered := FALSE;
	resettingState := 0;
	bagger.bagOpenFingers.RemovePower();
	bagger.vacuumBagOpen.StopVacuum();
	bagger.pressureBar.RemovePower();
	bagger.printer.Reset();
	bagger.bagDelivery.Reset();
	bagger.StartCycleRequest := FALSE;
	bagger.ReadyForProduct := FALSE;
	bagger.CurrentBagOpenRetryCount := 0;
	bagger.StartCycleRequest := FALSE;
	state := HEAD_STATES.Idle;
	sealAndSeparateSubState := SEAL_SEPARATE_STATES.Idle;
    releaseAndFeedSubState := RELEASE_FEED_STATES.Idle;
    bagOpenSubState := BAG_OPEN_ASSIST_STATES.Idle;
	cycleTimer.IN := FALSE;
	_abortingDone := TRUE;
END_IF

METHOD Aborted

_abortingDone := FALSE;

METHOD Clearing

IF NOT resetTriggered THEN
	bagger.pressureBar.Reset();

	_completingDone := FALSE;
	_holdingDone := FALSE;
	_resettingDone := FALSE;
	_startingDone := FALSE;
	_unholdingDone := FALSE;
	_stoppingDone := FALSE;
	resetTriggered := TRUE;
	_clearingDone := TRUE;
END_IF

// IF bagger.pressureBar.Ready THEN
// 	_clearingDone := TRUE;
// 	resetTriggered := FALSE;
// END_IF

METHOD Held

_holdingDone := FALSE;

METHOD Holding

_holdingDone := TRUE;

METHOD UnHolding

_unholdingDone := TRUE;

METHOD Complete

_completingDone := FALSE;

METHOD Completing

_completingDone := TRUE;

METHOD INTERNAL SetHeadState
VAR_INPUT
	newState : HEAD_STATES;
END_VAR

state := newState;
_logger.AddLogItem(CONCAT('Head State: ',TO_STRING(newState)));

METHOD INTERNAL SetSealSeparateState
VAR_INPUT
	newState : SEAL_SEPARATE_STATES;
END_VAR
VAR
	statePrefix : STRING;
END_VAR
sealAndSeparateSubState := newState;
statePrefix := CONCAT(TO_STRING(state), ' - ');
_logger.AddLogItem(CONCAT(statePrefix,TO_STRING(newState)));

METHOD INTERNAL SetReleaseFeedState
VAR_INPUT
	newState : RELEASE_FEED_STATES;
END_VAR

releaseAndFeedSubState := newState;
_logger.AddLogItem(CONCAT('Release/Feed State: ',TO_STRING(newState)));

METHOD INTERNAL SetBagOpenState
VAR_INPUT
	newState : BAG_OPEN_ASSIST_STATES;
END_VAR
VAR
	statePrefix : STRING;
END_VAR
bagOpenSubState := newState;
_logger.AddLogItem(CONCAT('Bag Open State: ',TO_STRING(newState)));

FUNCTION_BLOCK EM01_BaggerHead_Automode EXTENDS FB_PackMLStates
VAR_INPUT
	infeed : IEM00_Product_Infeed;
	discharge : IEM02_Discharge;
END_VAR
VAR_OUTPUT
	state : HEAD_STATES;
    sealAndSeparateSubState : SEAL_SEPARATE_STATES;
    releaseAndFeedSubState : RELEASE_FEED_STATES;
    bagOpenSubState : BAG_OPEN_ASSIST_STATES;
	currentBaggerState : STRING;
END_VAR
VAR
	cycleTimer : TON() := (PT := T#1000S);
	cycleTime : REAL;
	resetTriggered : BOOL;
	resettingState : INT;
	vacuumDwellTimer : TON;
END_VAR
VAR_IN_OUT
	bagger : EM01_BaggerHead;
END_VAR

//	Function Block: EM01_Bagger_Automode
//	Description: This is an implementation of a bagger in Auto Mode (normal operation) using the PackML standard.
//				 Each method is a PackML state.
//	Created by: Ben Hess
//	Created Date: Tuesday, March 26, 2019

METHOD Stopping

_stoppingDone := TRUE;

METHOD Stopped

_clearingDone := FALSE;
_stoppingDone := FALSE;
resetTriggered := FALSE;

METHOD Resetting

state := HEAD_STATES.Idle;
sealAndSeparateSubState := SEAL_SEPARATE_STATES.Idle;
releaseAndFeedSubState := RELEASE_FEED_STATES.Idle;
bagOpenSubState := BAG_OPEN_ASSIST_STATES.Idle;

CASE resettingState OF
	0:	// Clear PackML state bits and Home everything that needs homing
		_clearingDone := FALSE;
		_completingDone := FALSE;
		_holdingDone := FALSE;
		_resettingDone := FALSE;
		_startingDone := FALSE;
		_unholdingDone := FALSE;
		_stoppingDone := FALSE;

		vacuumDwellTimer.IN := FALSE;

		bagger.bagDelivery.Reset();
		HomeIfNeeded(bagger.pressureBar);
		HomeIfNeeded(bagger.sealFlatteners);
		resettingState := 1;

	1:	// Move everything into place to start machine
		IF CheckIfHomed(bagger.pressureBar) THEN
			PostHomeMoveIfNeeded(bagger.pressureBar);
			resettingState := 2;
		END_IF

	2:	// Once everything is moved into position and ready move on
		IF bagger.pressureBar.Ready OR NOT bagger.pressureBar.OptionActive THEN
			_resettingDone := TRUE;
		END_IF

END_CASE

METHOD Idle

_resettingDone := FALSE;
resettingState := 0;
resetTriggered := FALSE;

METHOD Starting

IF NOT _startingDone THEN
	bagger.pressureBar.Open();
	bagger.bagOpenFingers.ReleaseBag();
	bagger.sealFlatteners.ToBagFeed();
	_startingDone := TRUE;
END_IF

METHOD Executing

//	Method: EM01_Bagger_Automode.Executing()
//	Description: Executing is the state in which the machine is producing bags.  In this state, the bagger is homed and ready to initiate a cycle any time.
//				 In normal operation, the machine should be in this state most of the time
//				 The logic below is generic and coded to interfaces for each component
//	Created by: Ben Hess
//	Created Date: Tuesday, March 26, 2019

IF NOT __ISVALIDREF(bagger) THEN
	RETURN;
END_IF

// Clear starting done status because if we're here starting state is complete.
_startingDone := FALSE;

// Run Cycle timer for machine cycle
cycleTimer();
vacuumDwellTimer(PT := bagger.vacuumDwell);
// State machine for overall head states
CASE state OF
    HEAD_STATES.Idle :                              // Start cycle
                                                    IF bagger.StartCycleRequest THEN
														bagger.StartCycleRequest := FALSE;
														cycleTimer.IN := TRUE;
														_logger.AddLogItem('Cycle Started');
														SetHeadState(HEAD_STATES.SealAndSeparateBag);
													END_IF

													IF MoveRequested (bagger.pressureBar) THEN
														SetHeadState(HEAD_STATES.MovePassthrough);
													END_IF

	HEAD_STATES.MovePassthrough : 					//
													PostHomeMoveIfNeeded(bagger.pressureBar);
													SetHeadState(HEAD_STATES.MovingPassthrough);

    HEAD_STATES.MovingPassthrough :                 //
													IF NOT MoveRequested (bagger.pressureBar) THEN
														SetHeadState(HEAD_STATES.MovedPassthrough);
													END_IF

	HEAD_STATES.MovedPassthrough : 					//
													SetHeadState(HEAD_STATES.Idle);

    HEAD_STATES.SealAndSeparateBag :                // Begin Seal and Separate State machine
                                                    SetSealSeparateState(SEAL_SEPARATE_STATES.MoveJawIn);
													SetHeadState(HEAD_STATES.SealingAndSeparatingBag);

    HEAD_STATES.SealingAndSeparatingBag :          //
													IF sealAndSeparateSubState = SEAL_SEPARATE_STATES.Done THEN
														SetHeadState(HEAD_STATES.SealedAndSeparatedBag);
														SetSealSeparateState(SEAL_SEPARATE_STATES.Idle);
                                                    END_IF

    HEAD_STATES.SealedAndSeparatedBag :             //
													SetHeadState(HEAD_STATES.ReleaseAndFeedBag);

    HEAD_STATES.ReleaseAndFeedBag :                 // Open the jaw and release the bag
													SetReleaseFeedState(RELEASE_FEED_STATES.MoveJawOutAndFeedBag);
                                                    SetHeadState(HEAD_STATES.ReleasingAndFeedingBag);

    HEAD_STATES.ReleasingAndFeedingBag :            //
                                                    IF releaseAndFeedSubState = RELEASE_FEED_STATES.Done THEN
                                                        SetHeadState(HEAD_STATES.ReleasedAndFedBag);
                                                        SetReleaseFeedState(RELEASE_FEED_STATES.Idle);
                                                    END_IF

    HEAD_STATES.ReleasedAndFedBag :                 // Start opening bag if bag open assist is enabled, otherwise end cycle now
													IF bagger.bagOpenAssistEnabled THEN
														SetHeadState(HEAD_STATES.OpenBag);
													ELSE
														SetHeadState(HEAD_STATES.OpenedBag);
													END_IF

    HEAD_STATES.OpenBag :                            // Close jaw to grab the bag
                                                    SetBagOpenState(BAG_OPEN_ASSIST_STATES.MoveJawIn);
                                                    SetHeadState(HEAD_STATES.OpeningBag);

    HEAD_STATES.OpeningBag :                        // Open jaw and grab onto the bag.  Feed a new bag out if missed
                                                    IF bagOpenSubState = BAG_OPEN_ASSIST_STATES.Done THEN
                                                        SetHeadState(HEAD_STATES.OpenedBag);
                                                        SetBagOpenState(BAG_OPEN_ASSIST_STATES.Idle);
													ELSIF bagOpenSubState = BAG_OPEN_ASSIST_STATES.FeedNewBag THEN
														SetHeadState(HEAD_STATES.SealAndSeparateBag);
														SetBagOpenState(BAG_OPEN_ASSIST_STATES.Idle);
                                                    END_IF

    HEAD_STATES.OpenedBag :                         // End cycle
                                                    SetHeadState(HEAD_STATES.Idle);
													cycleTime := (TIME_TO_REAL(cycleTimer.ET) / 1000);
													cycleTimer.IN := FALSE;
													_logger.AddLogItem(CONCAT('Cycle Complete in ',TO_STRING(cycleTime)));

    //HEAD_STATES.Fault :

END_CASE

CASE sealAndSeparateSubState OF
    //SEAL_SEPARATE_STATES.Idle :

    SEAL_SEPARATE_STATES.MoveJawIn :                // Perform actions as enabled - close jaw and move flatteners out. If jaw is disabled then go right to reverse bag
                                                    IF bagger.sealFlatteners.OptionActive THEN
														bagger.sealFlatteners.ToSeal();
													END_IF
                                                    bagger.pressureBar.Close();
													SetSealSeparateState(SEAL_SEPARATE_STATES.MovingJawIn);

    SEAL_SEPARATE_STATES.MovingJawIn :              // If Jaw is in and flatteners out then move on
                                                   	IF (NOT bagger.sealFlatteners.OptionActive OR bagger.sealFlatteners.InPosition)
														AND bagger.pressureBar.IsFullyClosed THEN
															SetSealSeparateState(SEAL_SEPARATE_STATES.MovedJawIn);
                                                    END_IF

    SEAL_SEPARATE_STATES.MovedJawIn :               // Seal bag now if separate before seal option selected
													IF NOT bagger.separateBeforeSealEnabled THEN
														bagger.sealer.BeginSealing();
													END_IF
													SetSealSeparateState(SEAL_SEPARATE_STATES.ReverseBag);

    SEAL_SEPARATE_STATES.ReverseBag :               // Start reversing bag to seal
													bagger.bagDelivery.ReverseToSeparate();
													SetSealSeparateState(SEAL_SEPARATE_STATES.ReversingBag);

    SEAL_SEPARATE_STATES.ReversingBag :             //
                                                    IF bagger.bagDelivery.BagSeparated
														AND (bagger.sealer.SealComplete OR bagger.separateBeforeSealEnabled)
                                                        THEN
															SetSealSeparateState(SEAL_SEPARATE_STATES.Reversedbag);
                                                    END_IF

    SEAL_SEPARATE_STATES.Reversedbag :              //
                                                    IF bagger.separateBeforeSealEnabled THEN
														SetSealSeparateState(SEAL_SEPARATE_STATES.SealBag);
													ELSE
														SetSealSeparateState(SEAL_SEPARATE_STATES.Done);
													END_IF

	SEAL_SEPARATE_STATES.SealBag:
													bagger.sealer.BeginSealing();
													SetSealSeparateState(SEAL_SEPARATE_STATES.SealingBag);

	SEAL_SEPARATE_STATES.SealingBag:				//
													IF bagger.sealer.SealComplete THEN
														SetSealSeparateState(SEAL_SEPARATE_STATES.Done);
													END_IF

    //SEAL_SEPARATE_STATES.Done :                   //

    //SEAL_SEPARATE_STATES.Fault :					//
END_CASE

CASE releaseAndFeedSubState OF
    //RELEASE_FEED_STATES.Idle :                    //

    RELEASE_FEED_STATES.MoveJawOutAndFeedBag :
													bagger.bagOpenFingers.ReleaseBag();
													bagger.sealFlatteners.ToBagFeed();
													bagger.pressureBar.Open();

													discharge.TakeAwayBag(THIS^);
													releaseAndFeedSubState := RELEASE_FEED_STATES.WaitForOKFromDischarge;
													// If printer is enabled then perform printer operation of bag delivery, otherwise just feed new bag out.
													IF NOT bagger.printer.OptionActive THEN
														bagger.bagDelivery.FeedBagOut();
														SetReleaseFeedState(RELEASE_FEED_STATES.MovingJawOutAndFeedingBag);
													ELSE
														SetReleaseFeedState(RELEASE_FEED_STATES.WaitForPrinter);
													END_IF

    RELEASE_FEED_STATES.WaitForOKFromDischarge :   	// Wait for EM02 - Discharge to give OK to feed bag signal
													IF discharge.OKToFeedBag THEN
														IF NOT bagger.printer.OptionActive THEN
															bagger.bagDelivery.FeedBagOut();
															SetReleaseFeedState(RELEASE_FEED_STATES.MovingJawOutAndFeedingBag);
														ELSE
															SetReleaseFeedState(RELEASE_FEED_STATES.WaitForPrinter);
														END_IF
													END_IF

    RELEASE_FEED_STATES.WaitForPrinter :            // Data Ready means the printer has a label and we're all set to print
                                                    IF bagger.printer.HasLabel THEN
														SetReleaseFeedState(RELEASE_FEED_STATES.FeedToOffset);
                                                    END_IF

    RELEASE_FEED_STATES.FeedToOffset :              // Start feeding to the print offset
                                                    bagger.bagDelivery.FeedToPrintOffset();
													SetReleaseFeedState(RELEASE_FEED_STATES.FeedingToOffset);

    RELEASE_FEED_STATES.FeedingToOffset :            // Once offset done start printing
                                                    IF bagger.bagDelivery.ReadyForPrint THEN
														SetReleaseFeedState(RELEASE_FEED_STATES.StartPrinting);
                                                    END_IF

    RELEASE_FEED_STATES.StartPrinting :             // Printer starts print cycle and bag delivery starts moving at print speed
													bagger.printer.BeginPrinting();
													bagger.bagDelivery.FeedAtPrintSpeed();
													SetReleaseFeedState(RELEASE_FEED_STATES.Printing);

    //RELEASE_FEED_STATES.SendPrintSignal:            //

    RELEASE_FEED_STATES.Printing :                  // Wait for print to finish
                                                    IF bagger.printer.PrintDone THEN
														SetReleaseFeedState(RELEASE_FEED_STATES.StopPrinting);
                                                    END_IF

    RELEASE_FEED_STATES.StopPrinting :              // Tell bag delivery it's okay to feed out the rest of the bag and the printer that it can prep itself for the next print
                                                    bagger.bagDelivery.FeedBagOut();
													SetReleaseFeedState(RELEASE_FEED_STATES.MovingJawOutAndFeedingBag);

    RELEASE_FEED_STATES.MovingJawOutAndFeedingBag : //
													IF (bagger.sealFlatteners.InPosition OR NOT bagger.sealFlatteners.OptionActive)
                                                        AND bagger.pressureBar.IsFullyOpen
														AND bagger.bagDelivery.BagFeedDone
                                                        THEN
															SetReleaseFeedState(RELEASE_FEED_STATES.MovedJawOutAndFedBag);
                                                    END_IF

    RELEASE_FEED_STATES.MovedJawOutAndFedBag :
													SetReleaseFeedState(RELEASE_FEED_STATES.Done);
    //RELEASE_FEED_STATES.Done :
    //RELEASE_FEED_STATES.Fault :
END_CASE

CASE bagOpenSubState OF
    BAG_OPEN_ASSIST_STATES.Idle :                    //

    BAG_OPEN_ASSIST_STATES.MoveJawIn :                // Close jaw against bag. In the future we may also start vacuum here
                                                    bagger.pressureBar.Close();
													SetBagOpenState(BAG_OPEN_ASSIST_STATES.MovingJawIn);

    BAG_OPEN_ASSIST_STATES.MovingJawIn :            // Move on once jaw is closed
                                                    IF bagger.pressureBar.IsFullyClosed THEN
														IF bagger.vacuumBagOpen.OptionActive THEN
															bagger.vacuumBagOpen.StartVacuum();
														END_IF
														SetBagOpenState(BAG_OPEN_ASSIST_STATES.MovedJawIn);
                                                    END_IF

    BAG_OPEN_ASSIST_STATES.MovedJawIn :             // Hold onto the bag with vacuum to build suction
													vacuumDwellTimer.IN := TRUE;
													IF (vacuumDwellTimer.Q OR NOT bagger.vacuumBagOpen.OptionActive) THEN
														vacuumDwellTimer.IN := FALSE;
														SetBagOpenState(BAG_OPEN_ASSIST_STATES.MoveJawOut);
													END_IF

    BAG_OPEN_ASSIST_STATES.MoveJawOut :             // Open the jaw and move seal flatteners in and to bag holding
                                                    bagger.pressureBar.Open();
													SetBagOpenState(BAG_OPEN_ASSIST_STATES.MovingJawOutAndGrab);

    BAG_OPEN_ASSIST_STATES.MovingJawOutAndGrab :    	//
														IF bagger.bagOpenFingers.OptionActive THEN
															bagger.bagOpenFingers.GrabBag();
															IF bagger.bagOpenSensorEnabled THEN
																SetBagOpenState(BAG_OPEN_ASSIST_STATES.CheckForSuccessfulBagGrab);
															ELSE
																SetBagOpenState(BAG_OPEN_ASSIST_STATES.BagOpened);
															END_IF
														ELSE
															SetBagOpenState(BAG_OPEN_ASSIST_STATES.BagOpened);
														END_IF

	BAG_OPEN_ASSIST_STATES.CheckForSuccessfulBagGrab : 	//
														IF bagger.CurrentBagOpenRetryCount < bagger.bagOpenRetrySetting THEN
															IF bagger.bagOpenFingers.BagGrabbed THEN
																SetBagOpenState(BAG_OPEN_ASSIST_STATES.BagOpened);
															ELSIF bagger.bagOpenFingers.BagMissed THEN
																SetBagOpenState(BAG_OPEN_ASSIST_STATES.BagFailedToOpen);
															END_IF
														ELSE
															SetBagOpenState(BAG_OPEN_ASSIST_STATES.MovingJawOutAfterGrab);
														END_IF

	BAG_OPEN_ASSIST_STATES.BagFailedToOpen :			//
														bagger.bagOpenFingers.ReleaseBag();
														bagger.CurrentBagOpenRetryCount := bagger.CurrentBagOpenRetryCount + 1;
														IF bagger.CurrentBagOpenRetryCount < bagger.bagOpenRetrySetting THEN
															SetBagOpenState(BAG_OPEN_ASSIST_STATES.MoveJawIn);
														ELSE
															SetBagOpenState(BAG_OPEN_ASSIST_STATES.MovingJawOutAfterGrab);
															bagger.CurrentBagOpenRetryCount := 0;
															bagger.failedToOpenBag.Trigger();
														END_IF

	BAG_OPEN_ASSIST_STATES.BagOpened :					//
														bagger.vacuumBagOpen.StopVacuum();
                                                    	bagger.sealFlatteners.BagIsOpen();
														bagger.CurrentBagOpenRetryCount := 0;
// 														HMIData.bagsMade.Increment();
// 														HMIData.airFilterClean.Increment();
// 														HMIData.baggerCycles.Increment();
														SetBagOpenState(BAG_OPEN_ASSIST_STATES.MovingJawOutAfterGrab);

    BAG_OPEN_ASSIST_STATES.MovingJawOutAfterGrab :		//
														IF bagger.pressureBar.IsFullyOpen
															AND (bagger.sealFlatteners.InPosition OR NOT bagger.sealFlatteners.OptionActive)
															THEN
																SetBagOpenState(BAG_OPEN_ASSIST_STATES.MovedJawOut);
														END_IF

	BAG_OPEN_ASSIST_STATES.MovedJawOut :            	//

														SetBagOpenState(BAG_OPEN_ASSIST_STATES.Done);

	//BAG_OPEN_ASSIST_STATES.FeedNewBag :   				//

    //BAG_OPEN_ASSIST_STATES.Done :                    	//

    //BAG_OPEN_ASSIST_STATES.Fault :                    //

END_CASE

METHOD Aborting

IF NOT _abortingDone THEN
	_clearingDone := FALSE;
	_completingDone := FALSE;
	_holdingDone := FALSE;
	_resettingDone := FALSE;
	_startingDone := FALSE;
	_unholdingDone := FALSE;
	_stoppingDone := FALSE;
	resetTriggered := FALSE;
	resettingState := 0;
	bagger.bagOpenFingers.RemovePower();
	bagger.vacuumBagOpen.StopVacuum();
	bagger.pressureBar.RemovePower();
	bagger.printer.Reset();
	bagger.bagDelivery.Reset();
	bagger.StartCycleRequest := FALSE;
	bagger.ReadyForProduct := FALSE;
	bagger.CurrentBagOpenRetryCount := 0;
	bagger.StartCycleRequest := FALSE;
	state := HEAD_STATES.Idle;
	sealAndSeparateSubState := SEAL_SEPARATE_STATES.Idle;
    releaseAndFeedSubState := RELEASE_FEED_STATES.Idle;
    bagOpenSubState := BAG_OPEN_ASSIST_STATES.Idle;
	cycleTimer.IN := FALSE;
	_abortingDone := TRUE;
END_IF

METHOD Aborted

_abortingDone := FALSE;

METHOD Clearing

IF NOT resetTriggered THEN
	bagger.pressureBar.Reset();

	_completingDone := FALSE;
	_holdingDone := FALSE;
	_resettingDone := FALSE;
	_startingDone := FALSE;
	_unholdingDone := FALSE;
	_stoppingDone := FALSE;
	resetTriggered := TRUE;
	_clearingDone := TRUE;
END_IF

// IF bagger.pressureBar.Ready THEN
// 	_clearingDone := TRUE;
// 	resetTriggered := FALSE;
// END_IF

METHOD Held

_holdingDone := FALSE;

METHOD Holding

_holdingDone := TRUE;

METHOD UnHolding

_unholdingDone := TRUE;

METHOD Complete

_completingDone := FALSE;

METHOD Completing

_completingDone := TRUE;

METHOD INTERNAL SetHeadState
VAR_INPUT
	newState : HEAD_STATES;
END_VAR

state := newState;
_logger.AddLogItem(CONCAT('Head State: ',TO_STRING(newState)));

METHOD INTERNAL SetSealSeparateState
VAR_INPUT
	newState : SEAL_SEPARATE_STATES;
END_VAR
VAR
	statePrefix : STRING;
END_VAR
sealAndSeparateSubState := newState;
statePrefix := CONCAT(TO_STRING(state), ' - ');
_logger.AddLogItem(CONCAT(statePrefix,TO_STRING(newState)));

METHOD INTERNAL SetReleaseFeedState
VAR_INPUT
	newState : RELEASE_FEED_STATES;
END_VAR

releaseAndFeedSubState := newState;
_logger.AddLogItem(CONCAT('Release/Feed State: ',TO_STRING(newState)));

METHOD INTERNAL SetBagOpenState
VAR_INPUT
	newState : BAG_OPEN_ASSIST_STATES;
END_VAR
VAR
	statePrefix : STRING;
END_VAR
bagOpenSubState := newState;
_logger.AddLogItem(CONCAT('Bag Open State: ',TO_STRING(newState)));

(* ---- EM01_BaggerHead_MaintMode.st ---- *)
FUNCTION_BLOCK EM01_BaggerHead_MaintMode EXTENDS FB_PackMLStates
VAR_INPUT

END_VAR
VAR_OUTPUT
	state : HEAD_STATES;
    sealAndSeparateSubState : SEAL_SEPARATE_STATES;
    releaseAndFeedSubState : RELEASE_FEED_STATES;
    openBagSubState : BAG_OPEN_ASSIST_STATES;
END_VAR
VAR
	_beginCycleFromInfeeed : BOOL;
	_readyToAcceptProduct : BOOL;
	cycleTimer : TON() := (PT := T#1000S);
	cycleTime : REAL;
	bagOpenRetryCount : UINT;
	bagOpenRetrySetting : UINT := 3;
END_VAR
VAR_IN_OUT
	//modeManager : PACK_ML.UnitModeManager;
	bagger : EM01_BaggerHead;
END_VAR

//	Function Block: EM01_Bagger_Automode
//	Description: This is an implementation of a bagger in Auto Mode (normal operation) using the PackML standard.
//				 Each method is a PackML state.
//	Created by: Ben Hess
//	Created Date: Tuesday, March 26, 2019

METHOD Stopping

_stoppingDone := TRUE;

METHOD Stopped

_clearingDone := FALSE;

METHOD Resetting

state := HEAD_STATES.Idle;
sealAndSeparateSubState := SEAL_SEPARATE_STATES.Idle;
releaseAndFeedSubState := RELEASE_FEED_STATES.Idle;
openBagSubState := BAG_OPEN_ASSIST_STATES.Idle;
_resettingDone := TRUE;

METHOD Idle

_resettingDone := FALSE;

METHOD Starting

IF NOT _startingDone THEN
	bagger.pressureBar.Open();
	bagger.bagOpenFingers.ReleaseBag();
	bagger.sealFlatteners.ToBagFeed();
	_startingDone := TRUE;
END_IF

METHOD Executing

//	Method: EM01_Bagger_MaintMode.Executing()
//	Description: Executing is the state in which the machine is ready to accept "service commands".
//
//	Created by: Ben Hess
//	Created Date: Tuesday, March 27, 2019
_startingDone := FALSE;

METHOD Aborting

IF NOT _abortingDone THEN
	bagger.bagOpenFingers.RemovePower();
	bagger.vacuumBagOpen.StopVacuum();
	bagger.pressureBar.RemovePower();
	_abortingDone := TRUE;
END_IF

METHOD Aborted

_abortingDone := FALSE;

METHOD Clearing

_clearingDone := TRUE;

METHOD Held

_holdingDone := FALSE;

METHOD Holding

_holdingDone := TRUE;

METHOD UnHolding

_unholdingDone := TRUE;

METHOD Complete

_completingDone := FALSE;

METHOD Completing

_completingDone := TRUE;

(* ---- EM01_BaggerHead_Manager.st ---- *)
FUNCTION_BLOCK EM01_BaggerHead_Manager EXTENDS FB_PackMLStates
VAR_INPUT
	discharge : IEM02_Discharge;
END_VAR
VAR_OUTPUT
END_VAR
VAR
	activeBaggerMode : IPackMLStates;
	BaggerAutoMode : EM01_BaggerHead_Automode(name := 'Auto Mode Bagger');
	BaggerMaintMode : EM01_BaggerHead_MaintMode(name := 'Maintenance Mode Bagger');
	xInit : BOOL;
END_VAR
VAR_IN_OUT
	modeManager : PACK_ML.UnitModeManager;
	baggerHead : EM01_BaggerHead;
END_VAR

IF NOT xInit THEN
	BaggerAutoMode(bagger := baggerHead, discharge := discharge);
	BaggerMaintMode(bagger := baggerHead);
	xInit := TRUE;
END_IF

IF modeManager.ActiveUnitMode.Name = UN00_Globals.sAutomatic THEN
	activeBaggerMode := BaggerAutoMode;
ELSIF modeManager.ActiveUnitMode.Name = UN00_Globals.sMaintenance THEN
	activeBaggerMode := BaggerMaintMode;
END_IF

_abortingDone := activeBaggerMode.AbortingDone;
_clearingDone := activeBaggerMode.ClearingDone;
_completingDone := activeBaggerMode.CompletingDone;
_holdingDone := activeBaggerMode.HoldingDone;
_resettingDone := activeBaggerMode.ResettingDone;
_startingDone := activeBaggerMode.StartingDone;
_unholdingDone := activeBaggerMode.UnholdingDone;
_stoppingDone := activeBaggerMode.StoppingDone;

CASE modeManager.ActiveUnitMode.CurrentState OF
	PACK_ML.State.Stopped: 			activeBaggerMode.Stopped();
	PACK_ML.State.Aborted:			activeBaggerMode.Aborted();
	PACK_ML.State.Idle:				activeBaggerMode.Idle();
	PACK_ML.State.Held:				activeBaggerMode.Held();
	PACK_ML.State.Complete:			activeBaggerMode.Complete();
	PACK_ML.State.Resetting:		activeBaggerMode.Resetting();
	PACK_ML.State.Starting :		activeBaggerMode.Starting();
	PACK_ML.State.Execute :			activeBaggerMode.Executing();
	PACK_ML.State.Holding :			activeBaggerMode.Holding();
	PACK_ML.State.UnHolding :		activeBaggerMode.UnHolding();
	PACK_ML.State.Completing :		activeBaggerMode.Completing();
	PACK_ML.State.Aborting :		activeBaggerMode.Aborting();
	PACK_ML.State.Stopping:			activeBaggerMode.Stopping();
	PACK_ML.State.Clearing :		activeBaggerMode.Clearing();
END_CASE

FUNCTION_BLOCK EM01_BaggerHead_Manager EXTENDS FB_PackMLStates
VAR_INPUT
	discharge : IEM02_Discharge;
END_VAR
VAR_OUTPUT
END_VAR
VAR
	activeBaggerMode : IPackMLStates;
	BaggerAutoMode : EM01_BaggerHead_Automode(name := 'Auto Mode Bagger');
	BaggerMaintMode : EM01_BaggerHead_MaintMode(name := 'Maintenance Mode Bagger');
	xInit : BOOL;
END_VAR
VAR_IN_OUT
	modeManager : PACK_ML.UnitModeManager;
	baggerHead : EM01_BaggerHead;
END_VAR

IF NOT xInit THEN
	BaggerAutoMode(bagger := baggerHead, discharge := discharge);
	BaggerMaintMode(bagger := baggerHead);
	xInit := TRUE;
END_IF

IF modeManager.ActiveUnitMode.Name = UN00_Globals.sAutomatic THEN
	activeBaggerMode := BaggerAutoMode;
ELSIF modeManager.ActiveUnitMode.Name = UN00_Globals.sMaintenance THEN
	activeBaggerMode := BaggerMaintMode;
END_IF

_abortingDone := activeBaggerMode.AbortingDone;
_clearingDone := activeBaggerMode.ClearingDone;
_completingDone := activeBaggerMode.CompletingDone;
_holdingDone := activeBaggerMode.HoldingDone;
_resettingDone := activeBaggerMode.ResettingDone;
_startingDone := activeBaggerMode.StartingDone;
_unholdingDone := activeBaggerMode.UnholdingDone;
_stoppingDone := activeBaggerMode.StoppingDone;

CASE modeManager.ActiveUnitMode.CurrentState OF
	PACK_ML.State.Stopped: 			activeBaggerMode.Stopped();
	PACK_ML.State.Aborted:			activeBaggerMode.Aborted();
	PACK_ML.State.Idle:				activeBaggerMode.Idle();
	PACK_ML.State.Held:				activeBaggerMode.Held();
	PACK_ML.State.Complete:			activeBaggerMode.Complete();
	PACK_ML.State.Resetting:		activeBaggerMode.Resetting();
	PACK_ML.State.Starting :		activeBaggerMode.Starting();
	PACK_ML.State.Execute :			activeBaggerMode.Executing();
	PACK_ML.State.Holding :			activeBaggerMode.Holding();
	PACK_ML.State.UnHolding :		activeBaggerMode.UnHolding();
	PACK_ML.State.Completing :		activeBaggerMode.Completing();
	PACK_ML.State.Aborting :		activeBaggerMode.Aborting();
	PACK_ML.State.Stopping:			activeBaggerMode.Stopping();
	PACK_ML.State.Clearing :		activeBaggerMode.Clearing();
END_CASE

(* ---- EM02_Discharge.st ---- *)
FUNCTION_BLOCK EM02_Discharge EXTENDS FB_PackMLStates IMPLEMENTS IEM02_Discharge
VAR_INPUT
END_VAR
VAR_OUTPUT
END_VAR
VAR
END_VAR

{attribute 'monitoring' := 'call'}
PROPERTY OKToFeedBag : BOOL

{warning 'add property implementation'}
PROPERTY ReadyForProduct : BOOL

{warning 'add method implementation '}
METHOD TakeAwayBag
VAR_INPUT
		caller : IAllObjects;
END_VAR

FUNCTION_BLOCK EM02_Discharge EXTENDS FB_PackMLStates IMPLEMENTS IEM02_Discharge
VAR_INPUT
END_VAR
VAR_OUTPUT
END_VAR
VAR
END_VAR

{attribute 'monitoring' := 'call'}
PROPERTY OKToFeedBag : BOOL

{warning 'add property implementation'}
PROPERTY ReadyForProduct : BOOL

{warning 'add method implementation '}
METHOD TakeAwayBag
VAR_INPUT
		caller : IAllObjects;
END_VAR

(* ---- FB_AppliedMotionMotor.st ---- *)
FUNCTION_BLOCK FB_AppliedMotionMotor EXTENDS Sharp_Motion.Axis_REF
VAR_INPUT
END_VAR
VAR_OUTPUT
END_VAR
VAR
END_VAR

FUNCTION_BLOCK FB_AppliedMotionMotor EXTENDS Sharp_Motion.Axis_REF
VAR_INPUT
END_VAR
VAR_OUTPUT
END_VAR
VAR
END_VAR

(* ---- FB_BaseBagOpenFingers.st ---- *)
FUNCTION_BLOCK FB_BaseBagOpenFingers EXTENDS FB_BaseComponent IMPLEMENTS IBagOpenFingers
VAR_INPUT
	delayToGrabSetting : REAL;						// How long to wait afer a grab request to start moving fingers
	delayToCheckBagPresentSetting : REAL;			// How long to wait after grabbing bag to check if it is present
	delayToClearSetting : REAL;						// How long to wait after letting go of bag to call it clear of the pressure bar
END_VAR
VAR_OUTPUT
	grabCounter : FB_MachineCounter(name := CONCAT(_prefix, 'Grab Counter'));
	releaseCounter : FB_MachineCounter(name := CONCAT(_prefix, 'Release Counter'));
	missedCounter : FB_MachineCounter(name := CONCAT(_prefix, 'Missed Counter'));
END_VAR
VAR
	_grabBagRequest : BOOL;
	_releaseBagRequest : BOOL;
	_bagCleared : BOOL;
	_bagGrabbed : BOOL;
	_bagMissed : BOOL;
	delayToGrab : Standard.TON;
	delayToCheckBagPresent : Standard.TON;
	delayToClear : Standard.TON;
END_VAR
VAR_IN_OUT

END_VAR
SUPER^();
delayToGrab(IN := _grabBagRequest, PT := REAL_TO_TIME(delayToGrabSetting * 1000));
delayToCheckBagPresent(IN := delayToGrab.Q, PT := REAL_TO_TIME(delayToCheckBagPresentSetting * 1000));
delayToClear(IN := _releaseBagRequest, PT := REAL_TO_TIME(delayToClearSetting * 1000));

{attribute 'monitoring' := 'variable'}
PROPERTY BagCleared : BOOL

{attribute 'monitoring' := 'variable'}
PROPERTY BagGrabbed : BOOL

{attribute 'monitoring' := 'variable'}
PROPERTY BagMissed : BOOL

METHOD RemovePower
VAR_INPUT
END_VAR

_bagCleared := FALSE;
_bagGrabbed := FALSE;
_bagMissed := FALSE;
_grabBagRequest := FALSE;
_releaseBagRequest := FALSE;
_logger.AddLogItem(CONCAT(_prefix,' Remove Power Request'));

METHOD GrabBag

_bagCleared := FALSE;
_bagGrabbed := FALSE;
_bagMissed := FALSE;
_releaseBagRequest := FALSE;
_grabBagRequest := TRUE;
_logger.AddLogItem(CONCAT(_prefix,' Grab Bag Request'));

METHOD ReleaseBag

_bagCleared := FALSE;
_bagGrabbed := FALSE;
_bagMissed := FALSE;
_grabBagRequest := FALSE;
_releaseBagRequest := TRUE;
_logger.AddLogItem(CONCAT(_prefix,' Release Bag Request'));

FUNCTION_BLOCK FB_BaseBagOpenFingers EXTENDS FB_BaseComponent IMPLEMENTS IBagOpenFingers
VAR_INPUT
	delayToGrabSetting : REAL;						// How long to wait afer a grab request to start moving fingers
	delayToCheckBagPresentSetting : REAL;			// How long to wait after grabbing bag to check if it is present
	delayToClearSetting : REAL;						// How long to wait after letting go of bag to call it clear of the pressure bar
END_VAR
VAR_OUTPUT
	grabCounter : FB_MachineCounter(name := CONCAT(_prefix, 'Grab Counter'));
	releaseCounter : FB_MachineCounter(name := CONCAT(_prefix, 'Release Counter'));
	missedCounter : FB_MachineCounter(name := CONCAT(_prefix, 'Missed Counter'));
END_VAR
VAR
	_grabBagRequest : BOOL;
	_releaseBagRequest : BOOL;
	_bagCleared : BOOL;
	_bagGrabbed : BOOL;
	_bagMissed : BOOL;
	delayToGrab : Standard.TON;
	delayToCheckBagPresent : Standard.TON;
	delayToClear : Standard.TON;
END_VAR
VAR_IN_OUT

END_VAR
SUPER^();
delayToGrab(IN := _grabBagRequest, PT := REAL_TO_TIME(delayToGrabSetting * 1000));
delayToCheckBagPresent(IN := delayToGrab.Q, PT := REAL_TO_TIME(delayToCheckBagPresentSetting * 1000));
delayToClear(IN := _releaseBagRequest, PT := REAL_TO_TIME(delayToClearSetting * 1000));

{attribute 'monitoring' := 'variable'}
PROPERTY BagCleared : BOOL

{attribute 'monitoring' := 'variable'}
PROPERTY BagGrabbed : BOOL

{attribute 'monitoring' := 'variable'}
PROPERTY BagMissed : BOOL

METHOD RemovePower
VAR_INPUT
END_VAR

_bagCleared := FALSE;
_bagGrabbed := FALSE;
_bagMissed := FALSE;
_grabBagRequest := FALSE;
_releaseBagRequest := FALSE;
_logger.AddLogItem(CONCAT(_prefix,' Remove Power Request'));

METHOD GrabBag

_bagCleared := FALSE;
_bagGrabbed := FALSE;
_bagMissed := FALSE;
_releaseBagRequest := FALSE;
_grabBagRequest := TRUE;
_logger.AddLogItem(CONCAT(_prefix,' Grab Bag Request'));

METHOD ReleaseBag

_bagCleared := FALSE;
_bagGrabbed := FALSE;
_bagMissed := FALSE;
_grabBagRequest := FALSE;
_releaseBagRequest := TRUE;
_logger.AddLogItem(CONCAT(_prefix,' Release Bag Request'));

(* ---- FB_BaseBagOpenFingers_UnitTest.st ---- *)
{attribute 'test' := 'multitest'}
{attribute 'testcasename':='Base Bag Open Fingers'}
{attribute 'testcategory':='Machine Components'}
{attribute 'testcasetimeout':='5000'}

FUNCTION_BLOCK FB_BaseBagOpenFingers_UnitTest EXTENDS CBM.EtrigA
VAR_INPUT
	xGetTestInfo : BOOL;
    diTestCaseIndex : DINT;
END_VAR
VAR_OUTPUT
    sTestCaseName : STRING;
	sTestCaseCategories : STRING;
    diTestCaseCount : DINT;
    diTestCaseTimeout : DINT;
    sInfo : STRING;
	eError : UnitTestErrors;
    sError : STRING;
    eFailureMode : TM.FAILUREMODE;
END_VAR
VAR
	testee : FB_BaseBagOpenFingers(name := 'Test Base Bag Open Fingers');
	checkGrabTimer : Standard.TON;
	checkNotGrabTimer : Standard.TON;
	grabRequested : BOOL;
END_VAR

SUPER^();

{attribute 'hide'}
METHOD prvAbort : BOOL

SUPER^.prvAbort();

xAbortInProgress := FALSE;

{attribute 'hide'}
METHOD prvCyclicAction : BOOL

SUPER^.prvCyclicAction();
checkGrabTimer();
checkNotGrabTimer();
testee(
	delayToGrabSetting:= ,
	delayToCheckBagPresentSetting:= ,
	delayToClearSetting:= ,
	grabCounter=> ,
	releaseCounter=> ,
	missedCounter=> );
CASE diTestCaseIndex OF
    0: 	IF THIS^.xGetTestInfo THEN
            THIS^.sTestCaseName := 'Step 1: Check all statuses are clear on initialization';
            THIS^.sTestCaseCategories := 'Machine Components';
            THIS^.diTestCaseTimeout := 3000;
			xDone := TRUE;
		ELSE
			IF NOT testee.BagCleared
				AND NOT testee.BagGrabbed
				AND NOT testee.BagMissed
			THEN
				 xDone := TRUE;
			ELSE
				THIS^.sError := 'Status should be all false';
				xError := TRUE;
				eError := UnitTestErrors.Failure;
            	eFailureMode := TM.FAILUREMODE.AbortTestCase;
                iError := 1;
			END_IF
        END_IF
    1: 	IF THIS^.xGetTestInfo THEN
            THIS^.sTestCaseName := 'Step 2: Grab Bag and watch for BagGrabbed status';
            THIS^.sTestCaseCategories := 'Machine Components';
            THIS^.diTestCaseTimeout := 3000;
			xDone := TRUE;
		ELSE
			testee.delayToGrabSetting := 1.0;
			checkGrabTimer.IN := TRUE;
			checkGrabTimer.PT := T#1050MS;

			checkNotGrabTimer.IN := TRUE;
			checkNotGrabTimer.PT := T#900MS;

			IF NOT grabRequested THEN
				testee.GrabBag();
				grabRequested := TRUE;
			END_IF

			IF checkNotGrabTimer.Q THEN
				IF testee.delayToGrab.Q THEN
					THIS^.sError := 'Bag Grab Request occured too soon';
					xError := TRUE;
					eError := UnitTestErrors.Failure;
					eFailureMode := TM.FAILUREMODE.AbortTestCase;
					iError := 1;
				END_IF
				checkNotGrabTimer.IN := FALSE;
			ELSIF checkGrabTimer.Q THEN
				IF testee.delayToGrab.Q THEN
					xDone := TRUE;
				ELSE
					THIS^.sError := 'Bag Grab Timer not timed out';
					xError := TRUE;
					eError := UnitTestErrors.Failure;
					eFailureMode := TM.FAILUREMODE.AbortTestCase;
					iError := 1;
				END_IF
				checkGrabTimer.IN := FALSE;
			END_IF
        END_IF

    ELSE
        IF THIS^.diTestCaseIndex < 0 THEN
            THIS^.diTestCaseCount := 2;
            xDone := TRUE;
        ELSE
            THIS^.sInfo := 'Invalid test case index';
            eError := UnitTestErrors.Failure;
			xError := TRUE;
        END_IF
END_CASE

{attribute 'hide'}
METHOD prvResetOutputs : BOOL

SUPER^.prvResetOutputs();

sTestCaseName := '';
sTestCaseCategories := '';
diTestCaseCount := 0;
diTestCaseTimeout := 0;
sInfo := '';
sError := '';
eFailureMode := TM.FAILUREMODE.AbortTestCase;

{attribute 'hide'}
{warning 'Add method implementation '}
METHOD prvStart : BOOL

{attribute 'test' := 'multitest'}
{attribute 'testcasename':='Base Bag Open Fingers'}
{attribute 'testcategory':='Machine Components'}
{attribute 'testcasetimeout':='5000'}

FUNCTION_BLOCK FB_BaseBagOpenFingers_UnitTest EXTENDS CBM.EtrigA
VAR_INPUT
	xGetTestInfo : BOOL;
    diTestCaseIndex : DINT;
END_VAR
VAR_OUTPUT
    sTestCaseName : STRING;
	sTestCaseCategories : STRING;
    diTestCaseCount : DINT;
    diTestCaseTimeout : DINT;
    sInfo : STRING;
	eError : UnitTestErrors;
    sError : STRING;
    eFailureMode : TM.FAILUREMODE;
END_VAR
VAR
	testee : FB_BaseBagOpenFingers(name := 'Test Base Bag Open Fingers');
	checkGrabTimer : Standard.TON;
	checkNotGrabTimer : Standard.TON;
	grabRequested : BOOL;
END_VAR

SUPER^();

{attribute 'hide'}
METHOD prvAbort : BOOL

SUPER^.prvAbort();

xAbortInProgress := FALSE;

{attribute 'hide'}
METHOD prvCyclicAction : BOOL

SUPER^.prvCyclicAction();
checkGrabTimer();
checkNotGrabTimer();
testee(
	delayToGrabSetting:= ,
	delayToCheckBagPresentSetting:= ,
	delayToClearSetting:= ,
	grabCounter=> ,
	releaseCounter=> ,
	missedCounter=> );
CASE diTestCaseIndex OF
    0: 	IF THIS^.xGetTestInfo THEN
            THIS^.sTestCaseName := 'Step 1: Check all statuses are clear on initialization';
            THIS^.sTestCaseCategories := 'Machine Components';
            THIS^.diTestCaseTimeout := 3000;
			xDone := TRUE;
		ELSE
			IF NOT testee.BagCleared
				AND NOT testee.BagGrabbed
				AND NOT testee.BagMissed
			THEN
				 xDone := TRUE;
			ELSE
				THIS^.sError := 'Status should be all false';
				xError := TRUE;
				eError := UnitTestErrors.Failure;
            	eFailureMode := TM.FAILUREMODE.AbortTestCase;
                iError := 1;
			END_IF
        END_IF
    1: 	IF THIS^.xGetTestInfo THEN
            THIS^.sTestCaseName := 'Step 2: Grab Bag and watch for BagGrabbed status';
            THIS^.sTestCaseCategories := 'Machine Components';
            THIS^.diTestCaseTimeout := 3000;
			xDone := TRUE;
		ELSE
			testee.delayToGrabSetting := 1.0;
			checkGrabTimer.IN := TRUE;
			checkGrabTimer.PT := T#1050MS;

			checkNotGrabTimer.IN := TRUE;
			checkNotGrabTimer.PT := T#900MS;

			IF NOT grabRequested THEN
				testee.GrabBag();
				grabRequested := TRUE;
			END_IF

			IF checkNotGrabTimer.Q THEN
				IF testee.delayToGrab.Q THEN
					THIS^.sError := 'Bag Grab Request occured too soon';
					xError := TRUE;
					eError := UnitTestErrors.Failure;
					eFailureMode := TM.FAILUREMODE.AbortTestCase;
					iError := 1;
				END_IF
				checkNotGrabTimer.IN := FALSE;
			ELSIF checkGrabTimer.Q THEN
				IF testee.delayToGrab.Q THEN
					xDone := TRUE;
				ELSE
					THIS^.sError := 'Bag Grab Timer not timed out';
					xError := TRUE;
					eError := UnitTestErrors.Failure;
					eFailureMode := TM.FAILUREMODE.AbortTestCase;
					iError := 1;
				END_IF
				checkGrabTimer.IN := FALSE;
			END_IF
        END_IF

    ELSE
        IF THIS^.diTestCaseIndex < 0 THEN
            THIS^.diTestCaseCount := 2;
            xDone := TRUE;
        ELSE
            THIS^.sInfo := 'Invalid test case index';
            eError := UnitTestErrors.Failure;
			xError := TRUE;
        END_IF
END_CASE

{attribute 'hide'}
METHOD prvResetOutputs : BOOL

SUPER^.prvResetOutputs();

sTestCaseName := '';
sTestCaseCategories := '';
diTestCaseCount := 0;
diTestCaseTimeout := 0;
sInfo := '';
sError := '';
eFailureMode := TM.FAILUREMODE.AbortTestCase;

{attribute 'hide'}
{warning 'Add method implementation '}
METHOD prvStart : BOOL

(* ---- FB_BaseComponent.st ---- *)
FUNCTION_BLOCK FB_BaseComponent EXTENDS FB_BaseObject IMPLEMENTS IComponent, IMachineOption, IExecuteAutomatically
VAR_INPUT
END_VAR
VAR_OUTPUT

END_VAR
VAR
    _ready : BOOL;                    // Ready to be controlled
	_reset : BOOL;
	_optionActive : BOOL;
	_optionEnabled : BOOL;
	_optionInstalled : BOOL;
	enableONS : R_TRIG;
	resetONS : R_TRIG;
END_VAR

//	Function Block: BaseComponentFB
//	Description:  Extend this FB for each component as it contains the basic variables and logic that all components must share
//	In all extended FBs that have an Execute() method you must run the parent logic with SUPER^()
//	Created by: Ben Hess
//	Created Date: Friday, June 1, 2018

_optionActive := _optionEnabled AND _optionInstalled;

METHOD Execute
VAR_INPUT
END_VAR

_optionActive := _optionEnabled AND _optionInstalled;

{attribute 'monitoring' := 'variable'}
PROPERTY Ready : BOOL

METHOD Reset
VAR_INPUT
END_VAR

_reset := TRUE;

{attribute 'monitoring' := 'variable'}
PROPERTY OptionActive : BOOL

{attribute 'monitoring' := 'variable'}
PROPERTY OptionEnabled : BOOL

{attribute 'monitoring' := 'variable'}
PROPERTY OptionInstalled : BOOL

FUNCTION_BLOCK FB_BaseComponent EXTENDS FB_BaseObject IMPLEMENTS IComponent, IMachineOption, IExecuteAutomatically
VAR_INPUT
END_VAR
VAR_OUTPUT

END_VAR
VAR
    _ready : BOOL;                    // Ready to be controlled
	_reset : BOOL;
	_optionActive : BOOL;
	_optionEnabled : BOOL;
	_optionInstalled : BOOL;
	enableONS : R_TRIG;
	resetONS : R_TRIG;
END_VAR

//	Function Block: BaseComponentFB
//	Description:  Extend this FB for each component as it contains the basic variables and logic that all components must share
//	In all extended FBs that have an Execute() method you must run the parent logic with SUPER^()
//	Created by: Ben Hess
//	Created Date: Friday, June 1, 2018

_optionActive := _optionEnabled AND _optionInstalled;

METHOD Execute
VAR_INPUT
END_VAR

_optionActive := _optionEnabled AND _optionInstalled;

{attribute 'monitoring' := 'variable'}
PROPERTY Ready : BOOL

METHOD Reset
VAR_INPUT
END_VAR

_reset := TRUE;

{attribute 'monitoring' := 'variable'}
PROPERTY OptionActive : BOOL

{attribute 'monitoring' := 'variable'}
PROPERTY OptionEnabled : BOOL

{attribute 'monitoring' := 'variable'}
PROPERTY OptionInstalled : BOOL

(* ---- FB_BaseObject.st ---- *)
FUNCTION_BLOCK FB_BaseObject IMPLEMENTS IAllObjects, ILoggable
VAR_INPUT
END_VAR
VAR_OUTPUT
END_VAR
VAR
	_instanceName : STRING;			// Instance Name
	_prefix : STRING;
	_logger : IMachineLogger;
END_VAR

METHOD FB_Init : BOOL
VAR_INPUT
  bInitRetains : BOOL; // TRUE: the retain variables are initialized (reset warm / reset cold)
  bInCopyCode : BOOL;  // TRUE: the instance will be copied to the copy code afterward (online change)
  name : STRING;
END_VAR

_instanceName := name;
_prefix := CONCAT(name, ' ');
GlobalObjects.CollectionOfAllObjects.AddObject(THIS^);

{attribute 'monitoring' := 'variable'}
PROPERTY InstanceName : STRING

METHOD RegisterLogger
VAR_INPUT
	internalLogger : IMachineLogger;
END_VAR

_logger := internalLogger;

(* ---- FB_BasicPrinter.st ---- *)
FUNCTION_BLOCK FB_BasicPrinter EXTENDS FB_BaseComponent IMPLEMENTS IPrinter, ISimulateable
VAR_INPUT
	simulateIO : BOOL;
	printSpeed : UDINT;
	printLength : REAL;
END_VAR
VAR_OUTPUT
END_VAR
VAR
	_hasLabel : BOOL;
	_printDone : BOOL;
	_beginPrinting : BOOL;
	_printing : BOOL;
	_simulate : BOOL;
	state : INT;
END_VAR

SUPER^();

PROPERTY Simulate : BOOL

PROPERTY Printing : BOOL

PROPERTY HasLabel : BOOL

PROPERTY PrintDone : BOOL

METHOD BeginPrinting
_beginPrinting := TRUE;

FUNCTION_BLOCK FB_BasicPrinter EXTENDS FB_BaseComponent IMPLEMENTS IPrinter, ISimulateable
VAR_INPUT
	simulateIO : BOOL;
	printSpeed : UDINT;
	printLength : REAL;
END_VAR
VAR_OUTPUT
END_VAR
VAR
	_hasLabel : BOOL;
	_printDone : BOOL;
	_beginPrinting : BOOL;
	_printing : BOOL;
	_simulate : BOOL;
	state : INT;
END_VAR

SUPER^();

PROPERTY Simulate : BOOL

PROPERTY Printing : BOOL

PROPERTY HasLabel : BOOL

PROPERTY PrintDone : BOOL

METHOD BeginPrinting
_beginPrinting := TRUE;

(* ---- FB_BasicSealer.st ---- *)
FUNCTION_BLOCK FB_BasicSealer EXTENDS FB_BaseComponent IMPLEMENTS ISealer
VAR_INPUT
	simulateIO : BOOL;
	sealDwell : REFERENCE TO REAL;
END_VAR
VAR_OUTPUT
END_VAR
VAR
	_beginSealing : BOOL;
	beginSealingONS : FB_ONS;
	sealTimer : TON;
	_sealComplete : BOOL;
	sealActive : BOOL;
	state : INT;
	//beginSealing : FB_SimulatedFeedback(name := CONCAT(_prefix,'Begin Sealing'));
END_VAR

SUPER^();

beginSealingONS(CLK := _beginSealing);
sealTimer();

IF _reset THEN
	sealActive := FALSE;
	_sealComplete := FALSE;
	sealTimer.IN := FALSE;
	state := 0;
END_IF

CASE state OF

	0:	IF beginSealingONS.OSR THEN
			_beginSealing := FALSE;
			sealTimer.PT := TO_TIME(sealDwell * 1000.0);
			sealTimer.IN := TRUE;
			sealActive := TRUE;
			state := 1;
		END_IF

	1:	IF sealTimer.Q THEN
			sealTimer.IN := FALSE;
			_sealComplete := TRUE;
			sealActive := FALSE;
			state := 0;
		END_IF

	2: //

	3: //
END_CASE

{attribute 'monitoring' := 'variable'}
PROPERTY SealComplete : BOOL

METHOD BeginSealing

_beginSealing := TRUE;
sealTimer.IN := FALSE;
_sealComplete := FALSE;

(* ---- FB_CollectionHandlerActiveFaults.st ---- *)
FUNCTION_BLOCK FB_CollectionHandlerActiveFaults
VAR_INPUT
END_VAR
VAR
	Collection: ARRAY[0..GlobalObjects.MAX_FAULTS] OF IFault; // object array
	ObjNames   : ARRAY[0..GlobalObjects.MAX_FAULTS] OF STRING;
	_ArrayOver   : BOOL;
	_BadObj      : INT;
	_DupeObj   : INT;
	_OverObj   : INT;
	_TotalObj   : UINT;
END_VAR

VAR_OUTPUT
	faultActive : BOOL;
END_VAR
//	Function Block: FB_CollectionHandlerActiveFaults
//	Description: This collection handler adds and removes active faults to an array
//				 The add and remove methods are called from FB_Fault
//	Created by: Tom Jacobs
//	Created Date: Friday, September 7, 2018

METHOD AckAll
VAR_INPUT
END_VAR
VAR
	Cast : IFault;
	Fault : IFault;
	J : UINT;
END_VAR
// For each active fault in the array, ack it.
FOR J:= 0 TO _TotalObj - 1 DO
	IF (__QUERYINTERFACE(Collection[J], Cast)) THEN
		Cast.Ack();
	ELSE
		RETURN;
	END_IF
END_FOR

METHOD AddObject
VAR_INPUT
	Obj   : IFault;
END_VAR
VAR
	I   : UINT;
	J : UINT;
END_VAR
// Add the active fault to the array
FOR J:= 0 TO _TotalObj DO
	IF Collection[J] = Obj THEN
		// object pointer matches - it's already in here
		RETURN;
	END_IF
END_FOR

IF _TotalObj < GlobalObjects.MAX_FAULTS THEN
	Collection[_TotalObj]:= Obj;
	ObjNames[_TotalObj]:= Obj.InstanceName;
	_TotalObj:= _TotalObj + 1;
ELSE
	_ArrayOver:= TRUE;
	_OverObj:= _OverObj + 1;
END_IF
GlobalObjects.CollectionOfFaults.FaultUpdateForHMI();
faultActive := TRUE;

METHOD RemoveObject
VAR_INPUT
	Obj   : IFault;
END_VAR

VAR
	I   : UINT;
	J : UINT;
END_VAR

FOR I:= 0 TO _TotalObj DO
	IF Collection[I] = Obj THEN
		// object pointer matches - get rid of it
		FOR J := I TO _TotalObj DO
			Collection[J] := Collection[J+1];
			ObjNames[J]:= ObjNames[J+1];
		END_FOR
		_TotalObj := _TotalObj - 1;
		IF _TotalObj = 0 THEN
			GlobalObjects.CollectionOfFaults.FaultUpdateForHMI();
			faultActive := FALSE;
		END_IF
		RETURN;
	END_IF
END_FOR
